LIN {X 0,Y 297.033,Z 357.775,A -85,B 0,C 180,E1 -16432.036,E2 -16432.036} C_VEL
LIN {X 0,Y 297.41,Z 355.086,A -85,B 0,C 180,E1 -16433.79,E2 -16433.79} C_VEL
LIN {X 0,Y 297.936,Z 351.345,A -85,B 0,C 180,E1 -16435.645,E2 -16435.645} C_VEL
LIN {X 0,Y 298.718,Z 345.55,A -85,B 0,C 180,E1 -16437.879,E2 -16437.879} C_VEL
LIN {X 0,Y 299.838,Z 337.982,A -85,B 0,C 180,E1 -16440.135,E2 -16440.135} C_VEL
LIN {X 0,Y 301.105,Z 329.348,A -85,B 0,C 180,E1 -16442.173,E2 -16442.173} C_VEL
LIN {X 0,Y 302.519,Z 319.297,A -85,B 0,C 180,E1 -16444.054,E2 -16444.054} C_VEL
LIN {X 0,Y 303.821,Z 309.214,A -85,B 0,C 180,E1 -16445.577,E2 -16445.577} C_VEL
LIN {X 0,Y 305.13,Z 297.791,A -85,B 0,C 180,E1 -16446.949,E2 -16446.949} C_VEL
LIN {X 0,Y 305.794,Z 291.875,A -85,B 0,C 180,E1 -16447.538,E2 -16447.538} C_VEL
LIN {X 0,Y 304.033,Z 282.592,A -85,B 0,C 180,E1 -16448.5,E2 -16448.5} C_VEL
LIN {X 0,Y 300.885,Z 269.635,A -85,B 0,C 180,E1 -16449.625,E2 -16449.625} C_VEL
LIN {X 0,Y 297.457,Z 257.519,A -85,B 0,C 180,E1 -16450.469,E2 -16450.469} C_VEL
LIN {X 0,Y 297.653,Z 253.673,A -85,B 0,C 180,E1 -16454.947,E2 -16454.947} C_VEL
LIN {X 0,Y 297.831,Z 251.39,A -85,B 0,C 180,E1 -16457.739,E2 -16457.739} C_VEL
LIN {X 0,Y 298.536,Z 251.297,A -85,B 0,C 180,E1 -16461.881,E2 -16461.881} C_VEL
LIN {X 0,Y 298.622,Z 251.286,A -85,B 0,C 180,E1 -16464.599,E2 -16464.599} C_VEL
LIN {X 0,Y 298.914,Z 251.25,A -85,B 0,C 180,E1 -16468.654,E2 -16468.654} C_VEL
LIN {X 0,Y 298.91,Z 251.253,A -85,B 0,C 180,E1 -16471.348,E2 -16471.348} C_VEL
LIN {X 0,Y 298.783,Z 251.266,A -85,B 0,C 180,E1 -16476.755,E2 -16476.755} C_VEL
LIN {X 0,Y 298.666,Z 251.281,A -85,B 0,C 180,E1 -16479.482,E2 -16479.482} C_VEL
LIN {X 0,Y 298.539,Z 251.297,A -85,B 0,C 180,E1 -16483.617,E2 -16483.617} C_VEL
LIN {X 0,Y 298.536,Z 251.297,A -85,B 0,C 180,E1 -16486.41,E2 -16486.41} C_VEL
LIN {X 0,Y 298.552,Z 251.294,A -85,B 0,C 180,E1 -16489.685,E2 -16489.685} C_VEL
LIN {X 0,Y 298.477,Z 251.304,A -85,B 0,C 180,E1 -16493.597,E2 -16493.597} C_VEL
LIN {X 0,Y 298.48,Z 251.305,A -85,B 0,C 180,E1 -16496.576,E2 -16496.576} C_VEL
LIN {X 0,Y 298.409,Z 251.311,A -85,B 0,C 180,E1 -16499.643,E2 -16499.643} C_VEL
LIN {X 0,Y 298.384,Z 251.319,A -85,B 0,C 180,E1 -16502.802,E2 -16502.802} C_VEL
LIN {X 0,Y 298.456,Z 251.308,A -85,B 0,C 180,E1 -16506.815,E2 -16506.815} C_VEL
LIN {X 0,Y 298.445,Z 251.307,A -85,B 0,C 180,E1 -16511.252,E2 -16511.252} C_VEL
LIN {X 0,Y 298.481,Z 251.302,A -85,B 0,C 180,E1 -16515.063,E2 -16515.063} C_VEL
LIN {X 0,Y 298.449,Z 251.306,A -85,B 0,C 180,E1 -16518.899,E2 -16518.899} C_VEL
LIN {X 0,Y 298.465,Z 251.304,A -85,B 0,C 180,E1 -16523.189,E2 -16523.189} C_VEL
LIN {X 0,Y 298.393,Z 251.312,A -85,B 0,C 180,E1 -16527.203,E2 -16527.203} C_VEL
LIN {X 0,Y 298.428,Z 251.309,A -85,B 0,C 180,E1 -16530.617,E2 -16530.617} C_VEL
LIN {X 0,Y 298.481,Z 251.302,A -85,B 0,C 180,E1 -16533.477,E2 -16533.477} C_VEL
LIN {X 0,Y 298.432,Z 251.309,A -85,B 0,C 180,E1 -16536.7,E2 -16536.7} C_VEL
LIN {X 0,Y 298.538,Z 251.293,A -85,B 0,C 180,E1 -16540.759,E2 -16540.759} C_VEL
LIN {X 0,Y 298.593,Z 251.287,A -85,B 0,C 180,E1 -16544.997,E2 -16544.997} C_VEL
LIN {X 0,Y 298.592,Z 251.289,A -85,B 0,C 180,E1 -16549.149,E2 -16549.149} C_VEL
LIN {X 0,Y 298.719,Z 251.277,A -85,B 0,C 180,E1 -16551.887,E2 -16551.887} C_VEL
LIN {X 0,Y 298.655,Z 251.278,A -85,B 0,C 180,E1 -16554.609,E2 -16554.609} C_VEL
LIN {X 0,Y 297.958,Z 251.369,A -85,B 0,C 180,E1 -16555.736,E2 -16555.736} C_VEL
LIN {X 0,Y 295.263,Z 251.704,A -85,B 0,C 180,E1 -16557.578,E2 -16557.578} C_VEL
LIN {X 0,Y 292.236,Z 252.085,A -85,B 0,C 180,E1 -16559.836,E2 -16559.836} C_VEL
LIN {X 0,Y 291.913,Z 252.12,A -85,B 0,C 180,E1 -16560.613,E2 -16560.613} C_VEL
LIN {X 0,Y 291.789,Z 252.136,A -85,B 0,C 180,E1 -16562.763,E2 -16562.763} C_VEL
LIN {X 0,Y 291.7,Z 252.144,A -85,B 0,C 180,E1 -16566.921,E2 -16566.921} C_VEL
LIN {X 0,Y 291.573,Z 252.167,A -85,B 0,C 180,E1 -16569.716,E2 -16569.716} C_VEL
LIN {X 0,Y 291.528,Z 252.169,A -85,B 0,C 180,E1 -16573.952,E2 -16573.952} C_VEL
LIN {X 0,Y 291.493,Z 252.171,A -85,B 0,C 180,E1 -16576.82,E2 -16576.82} C_VEL
LIN {X 0,Y 291.457,Z 252.179,A -85,B 0,C 180,E1 -16579.877,E2 -16579.877} C_VEL
LIN {X 0,Y 291.406,Z 252.184,A -85,B 0,C 180,E1 -16584.207,E2 -16584.207} C_VEL
LIN {X 0,Y 291.426,Z 252.186,A -85,B 0,C 180,E1 -16587.273,E2 -16587.273} C_VEL
LIN {X 0,Y 291.342,Z 252.192,A -85,B 0,C 180,E1 -16590.439,E2 -16590.439} C_VEL
LIN {X 0,Y 291.352,Z 252.192,A -85,B 0,C 180,E1 -16593.7,E2 -16593.7} C_VEL
LIN {X 0,Y 291.384,Z 252.191,A -85,B 0,C 180,E1 -16597.255,E2 -16597.255} C_VEL
LIN {X 0,Y 291.388,Z 252.232,A -85,B 0,C 180,E1 -16599.836,E2 -16599.836} C_VEL
LIN {X 0,Y 292.258,Z 257.11,A -85,B 0,C 180,E1 -16603.828,E2 -16603.828} C_VEL
LIN {X 0,Y 293.264,Z 262.494,A -85,B 0,C 180,E1 -16607.982,E2 -16607.982} C_VEL
LIN {X 0,Y 294.099,Z 267.529,A -85,B 0,C 180,E1 -16611.587,E2 -16611.587} C_VEL
LIN {X 0,Y 294.17,Z 270.073,A -85,B 0,C 180,E1 -16613.324,E2 -16613.324} C_VEL
LIN {X 0,Y 293.683,Z 273.84,A -85,B 0,C 180,E1 -16615.78,E2 -16615.78} C_VEL
LIN {X 0,Y 292.608,Z 280.296,A -85,B 0,C 180,E1 -16619.848,E2 -16619.848} C_VEL
LIN {X 0,Y 291.71,Z 286.456,A -85,B 0,C 180,E1 -16623.641,E2 -16623.641} C_VEL
LIN {X 0,Y 291.315,Z 289.802,A -85,B 0,C 180,E1 -16625.668,E2 -16625.668} C_VEL
LIN {X 0,Y 293.73,Z 303.932,A -85,B 0,C 180,E1 -16626.515,E2 -16626.515} C_VEL
LIN {X 0,Y 295.445,Z 316.454,A -85,B 0,C 180,E1 -16627.509,E2 -16627.509} C_VEL
LIN {X 0,Y 296.597,Z 328.112,A -85,B 0,C 180,E1 -16628.657,E2 -16628.657} C_VEL
LIN {X 0,Y 297.147,Z 337.485,A -85,B 0,C 180,E1 -16629.762,E2 -16629.762} C_VEL
LIN {X 0,Y 295.444,Z 348.79,A -85,B 0,C 180,E1 -16631.268,E2 -16631.268} C_VEL
LIN {X 0,Y 294.12,Z 358.492,A -85,B 0,C 180,E1 -16632.906,E2 -16632.906} C_VEL
LIN {X 0,Y 292.817,Z 367.103,A -85,B 0,C 180,E1 -16634.691,E2 -16634.691} C_VEL
LIN {X 0,Y 291.583,Z 375.192,A -85,B 0,C 180,E1 -16636.762,E2 -16636.762} C_VEL
LIN {X 0,Y 290.672,Z 381.694,A -85,B 0,C 180,E1 -16638.846,E2 -16638.846} C_VEL
LIN {X 0,Y 290.061,Z 386.848,A -85,B 0,C 180,E1 -16640.938,E2 -16640.938} C_VEL
LIN {X 0,Y 289.731,Z 390.835,A -85,B 0,C 180,E1 -16643.033,E2 -16643.033} C_VEL
LIN {X 0,Y 289.652,Z 392.878,A -85,B 0,C 180,E1 -16644.43,E2 -16644.43} C_VEL
LIN {X 0,Y 289.605,Z 394.493,A -85,B 0,C 180,E1 -16645.824,E2 -16645.824} C_VEL
LIN {X 0,Y 289.561,Z 395.692,A -85,B 0,C 180,E1 -16647.217,E2 -16647.217} C_VEL
LIN {X 0,Y 289.583,Z 396.449,A -85,B 0,C 180,E1 -16648.609,E2 -16648.609} C_VEL
LIN {X 0,Y 289.691,Z 396.79,A -85,B 0,C 180,E1 -16649.999,E2 -16649.999} C_VEL
LIN {X 0,Y 289.554,Z 396.262,A -85,B 0,C 180,E1 -16652.782,E2 -16652.782} C_VEL
LIN {X 0,Y 289.565,Z 395.378,A -85,B 0,C 180,E1 -16654.175,E2 -16654.175} C_VEL
LIN {X 0,Y 289.636,Z 393.816,A -85,B 0,C 180,E1 -16655.797,E2 -16655.797} C_VEL
LIN {X 0,Y 289.911,Z 390.214,A -85,B 0,C 180,E1 -16658.363,E2 -16658.363} C_VEL
LIN {X 0,Y 290.452,Z 386.109,A -85,B 0,C 180,E1 -16660.455,E2 -16660.455} C_VEL
LIN {X 0,Y 291.419,Z 379.871,A -85,B 0,C 180,E1 -16662.889,E2 -16662.889} C_VEL
LIN {X 0,Y 292.767,Z 373.132,A -85,B 0,C 180,E1 -16664.954,E2 -16664.954} C_VEL
LIN {X 0,Y 294.385,Z 364.544,A -85,B 0,C 180,E1 -16667.073,E2 -16667.073} C_VEL
LIN {X 0,Y 295.779,Z 356.408,A -85,B 0,C 180,E1 -16668.709,E2 -16668.709} C_VEL
LIN {X 0,Y 297.772,Z 346.112,A -85,B 0,C 180,E1 -16670.372,E2 -16670.372} C_VEL
LIN {X 0,Y 298.85,Z 338.795,A -85,B 0,C 180,E1 -16671.377,E2 -16671.377} C_VEL
LIN {X 0,Y 298.679,Z 327.3,A -85,B 0,C 180,E1 -16672.824,E2 -16672.824} C_VEL
LIN {X 0,Y 297.839,Z 315.601,A -85,B 0,C 180,E1 -16674.077,E2 -16674.077} C_VEL
LIN {X 0,Y 295.706,Z 302.829,A -85,B 0,C 180,E1 -16675.289,E2 -16675.289} C_VEL
LIN {X 0,Y 292.498,Z 290.386,A -85,B 0,C 180,E1 -16676.342,E2 -16676.342} C_VEL
LIN {X 0,Y 291.804,Z 287.336,A -85,B 0,C 180,E1 -16676.591,E2 -16676.591} C_VEL
LIN {X 0,Y 292.734,Z 281.581,A -85,B 0,C 180,E1 -16680.275,E2 -16680.275} C_VEL
LIN {X 0,Y 293.839,Z 275.714,A -85,B 0,C 180,E1 -16684.198,E2 -16684.198} C_VEL
LIN {X 0,Y 294.467,Z 272.269,A -85,B 0,C 180,E1 -16686.631,E2 -16686.631} C_VEL
LIN {X 0,Y 294.397,Z 268.901,A -85,B 0,C 180,E1 -16689.232,E2 -16689.232} C_VEL
LIN {X 0,Y 293.583,Z 264.391,A -85,B 0,C 180,E1 -16693.101,E2 -16693.101} C_VEL
LIN {X 0,Y 292.737,Z 259.678,A -85,B 0,C 180,E1 -16697.759,E2 -16697.759} C_VEL
LIN {X 0,Y 292.15,Z 256.569,A -85,B 0,C 180,E1 -16701.282,E2 -16701.282} C_VEL
LIN {X 0,Y 291.668,Z 253.761,A -85,B 0,C 180,E1 -16705.009,E2 -16705.009} C_VEL
LIN {X 0,Y 291.345,Z 252.195,A -85,B 0,C 180,E1 -16707.594,E2 -16707.594} C_VEL
LIN {X 0,Y 291.382,Z 252.187,A -85,B 0,C 180,E1 -16711.156,E2 -16711.156} C_VEL
LIN {X 0,Y 291.417,Z 252.186,A -85,B 0,C 180,E1 -16714.27,E2 -16714.27} C_VEL
LIN {X 0,Y 291.381,Z 252.185,A -85,B 0,C 180,E1 -16717.297,E2 -16717.297} C_VEL
LIN {X 0,Y 291.457,Z 252.176,A -85,B 0,C 180,E1 -16720.268,E2 -16720.268} C_VEL
LIN {X 0,Y 291.554,Z 252.164,A -85,B 0,C 180,E1 -16724.621,E2 -16724.621} C_VEL
LIN {X 0,Y 291.535,Z 252.168,A -85,B 0,C 180,E1 -16728.878,E2 -16728.878} C_VEL
LIN {X 0,Y 291.706,Z 252.146,A -85,B 0,C 180,E1 -16731.686,E2 -16731.686} C_VEL
LIN {X 0,Y 291.629,Z 252.16,A -85,B 0,C 180,E1 -16734.466,E2 -16734.466} C_VEL
LIN {X 0,Y 291.888,Z 252.129,A -85,B 0,C 180,E1 -16738.618,E2 -16738.618} C_VEL
LIN {X 0,Y 291.887,Z 252.126,A -85,B 0,C 180,E1 -16741.377,E2 -16741.377} C_VEL
LIN {X 0,Y 291.644,Z 252.357,A -85,B 0,C 180,E1 -16745.529,E2 -16745.529} C_VEL
LIN {X 0,Y 291.961,Z 253.705,A -85,B 0,C 180,E1 -16748.302,E2 -16748.302} C_VEL
LIN {X 0,Y 291.794,Z 256.101,A -85,B 0,C 180,E1 -16752.517,E2 -16752.517} C_VEL
LIN {X 0,Y 291.598,Z 257.897,A -85,B 0,C 180,E1 -16755.41,E2 -16755.41} C_VEL
LIN {X 0,Y 291.238,Z 260.78,A -85,B 0,C 180,E1 -16759.761,E2 -16759.761} C_VEL
LIN {X 0,Y 291.188,Z 261.337,A -85,B 0,C 180,E1 -16760.482,E2 -16760.482} C_VEL
LIN {X 0,Y 292.271,Z 264.393,A -85,B 0,C 180,E1 -16760.771,E2 -16760.771} C_VEL
LIN {X 0,Y 296.77,Z 275.63,A -85,B 0,C 180,E1 -16762.011,E2 -16762.011} C_VEL
LIN {X 0,Y 300.031,Z 286.603,A -85,B 0,C 180,E1 -16763.281,E2 -16763.281} C_VEL
LIN {X 0,Y 302.16,Z 296.713,A -85,B 0,C 180,E1 -16764.564,E2 -16764.564} C_VEL
LIN {X 0,Y 302.165,Z 299.449,A -85,B 0,C 180,E1 -16764.896,E2 -16764.896} C_VEL
LIN {X 0,Y 300.604,Z 309.905,A -85,B 0,C 180,E1 -16766.165,E2 -16766.165} C_VEL
LIN {X 0,Y 298.7,Z 320.617,A -85,B 0,C 180,E1 -16767.782,E2 -16767.782} C_VEL
LIN {X 0,Y 296.859,Z 330.143,A -85,B 0,C 180,E1 -16769.601,E2 -16769.601} C_VEL
LIN {X 0,Y 295.135,Z 338.506,A -85,B 0,C 180,E1 -16771.59,E2 -16771.59} C_VEL
LIN {X 0,Y 293.541,Z 345.871,A -85,B 0,C 180,E1 -16773.821,E2 -16773.821} C_VEL
LIN {X 0,Y 292.187,Z 351.715,A -85,B 0,C 180,E1 -16776.103,E2 -16776.103} C_VEL
LIN {X 0,Y 291.343,Z 355.527,A -85,B 0,C 180,E1 -16778.041,E2 -16778.041} C_VEL
LIN {X 0,Y 290.847,Z 357.596,A -85,B 0,C 180,E1 -16779.355,E2 -16779.355} C_VEL
LIN {X 0,Y 290.279,Z 359.966,A -85,B 0,C 180,E1 -16781.364,E2 -16781.364} C_VEL
LIN {X 0,Y 289.86,Z 361.443,A -85,B 0,C 180,E1 -16783.334,E2 -16783.334} C_VEL
LIN {X 0,Y 289.632,Z 362.114,A -85,B 0,C 180,E1 -16785.277,E2 -16785.277} C_VEL
LIN {X 0,Y 289.486,Z 362.005,A -85,B 0,C 180,E1 -16787.176,E2 -16787.176} C_VEL
LIN {X 0,Y 289.573,Z 361.135,A -85,B 0,C 180,E1 -16789.059,E2 -16789.059} C_VEL
LIN {X 0,Y 289.921,Z 358.545,A -85,B 0,C 180,E1 -16791.82,E2 -16791.82} C_VEL
LIN {X 0,Y 290.317,Z 355.666,A -85,B 0,C 180,E1 -16793.779,E2 -16793.779} C_VEL
LIN {X 0,Y 291.051,Z 350.63,A -85,B 0,C 180,E1 -16796.264,E2 -16796.264} C_VEL
LIN {X 0,Y 291.846,Z 344.907,A -85,B 0,C 180,E1 -16798.416,E2 -16798.416} C_VEL
LIN {X 0,Y 293.013,Z 337.475,A -85,B 0,C 180,E1 -16800.62,E2 -16800.62} C_VEL
LIN {X 0,Y 294.287,Z 328.968,A -85,B 0,C 180,E1 -16802.618,E2 -16802.618} C_VEL
LIN {X 0,Y 295.782,Z 318.782,A -85,B 0,C 180,E1 -16804.536,E2 -16804.536} C_VEL
LIN {X 0,Y 297.178,Z 308.303,A -85,B 0,C 180,E1 -16806.11,E2 -16806.11} C_VEL
LIN {X 0,Y 298.568,Z 296.305,A -85,B 0,C 180,E1 -16807.538,E2 -16807.538} C_VEL
LIN {X 0,Y 298.958,Z 292.63,A -85,B 0,C 180,E1 -16807.907,E2 -16807.907} C_VEL
LIN {X 0,Y 296.84,Z 282.192,A -85,B 0,C 180,E1 -16809.017,E2 -16809.017} C_VEL
LIN {X 0,Y 293.698,Z 269.415,A -85,B 0,C 180,E1 -16810.149,E2 -16810.149} C_VEL
LIN {X 0,Y 290.453,Z 257.903,A -85,B 0,C 180,E1 -16810.984,E2 -16810.984} C_VEL
LIN {X 0,Y 290.637,Z 254.275,A -85,B 0,C 180,E1 -16815.284,E2 -16815.284} C_VEL
LIN {X 0,Y 290.749,Z 252.496,A -85,B 0,C 180,E1 -16817.436,E2 -16817.436} C_VEL
LIN {X 0,Y 291.433,Z 252.185,A -85,B 0,C 180,E1 -16821.367,E2 -16821.367} C_VEL
LIN {X 0,Y 291.617,Z 252.161,A -85,B 0,C 180,E1 -16823.08,E2 -16823.08} C_VEL
LIN {X 0,Y 291.783,Z 252.142,A -85,B 0,C 180,E1 -16827.24,E2 -16827.24} C_VEL
LIN {X 0,Y 291.965,Z 252.115,A -85,B 0,C 180,E1 -16830.001,E2 -16830.001} C_VEL
LIN {X 0,Y 291.776,Z 252.139,A -85,B 0,C 180,E1 -16832.762,E2 -16832.762} C_VEL
LIN {X 0,Y 291.732,Z 252.146,A -85,B 0,C 180,E1 -16836.919,E2 -16836.919} C_VEL
LIN {X 0,Y 291.615,Z 252.159,A -85,B 0,C 180,E1 -16839.713,E2 -16839.713} C_VEL
LIN {X 0,Y 291.509,Z 252.172,A -85,B 0,C 180,E1 -16843.952,E2 -16843.952} C_VEL
LIN {X 0,Y 291.475,Z 252.18,A -85,B 0,C 180,E1 -16846.819,E2 -16846.819} C_VEL
LIN {X 0,Y 291.482,Z 252.174,A -85,B 0,C 180,E1 -16849.901,E2 -16849.901} C_VEL
LIN {X 0,Y 291.425,Z 252.183,A -85,B 0,C 180,E1 -16854.204,E2 -16854.204} C_VEL
LIN {X 0,Y 291.414,Z 252.183,A -85,B 0,C 180,E1 -16857.273,E2 -16857.273} C_VEL
LIN {X 0,Y 291.326,Z 252.196,A -85,B 0,C 180,E1 -16860.439,E2 -16860.439} C_VEL
LIN {X 0,Y 291.334,Z 252.192,A -85,B 0,C 180,E1 -16863.7,E2 -16863.7} C_VEL
LIN {X 0,Y 291.389,Z 252.185,A -85,B 0,C 180,E1 -16867.262,E2 -16867.262} C_VEL
LIN {X 0,Y 291.392,Z 252.19,A -85,B 0,C 180,E1 -16870.633,E2 -16870.633} C_VEL
LIN {X 0,Y 291.399,Z 252.188,A -85,B 0,C 180,E1 -16874.382,E2 -16874.382} C_VEL
LIN {X 0,Y 291.384,Z 252.187,A -85,B 0,C 180,E1 -16878.392,E2 -16878.392} C_VEL
LIN {X 0,Y 291.381,Z 252.186,A -85,B 0,C 180,E1 -16881.167,E2 -16881.167} C_VEL
LIN {X 0,Y 291.381,Z 252.189,A -85,B 0,C 180,E1 -16884.632,E2 -16884.632} C_VEL
LIN {X 0,Y 291.371,Z 252.188,A -85,B 0,C 180,E1 -16887.954,E2 -16887.954} C_VEL
LIN {X 0,Y 291.378,Z 252.184,A -85,B 0,C 180,E1 -16891.161,E2 -16891.161} C_VEL
LIN {X 0,Y 291.414,Z 252.187,A -85,B 0,C 180,E1 -16894.275,E2 -16894.275} C_VEL
LIN {X 0,Y 291.379,Z 252.187,A -85,B 0,C 180,E1 -16897.302,E2 -16897.302} C_VEL
LIN {X 0,Y 291.457,Z 252.178,A -85,B 0,C 180,E1 -16900.273,E2 -16900.273} C_VEL
LIN {X 0,Y 291.555,Z 252.164,A -85,B 0,C 180,E1 -16904.626,E2 -16904.626} C_VEL
LIN {X 0,Y 291.536,Z 252.167,A -85,B 0,C 180,E1 -16908.883,E2 -16908.883} C_VEL
LIN {X 0,Y 291.669,Z 252.154,A -85,B 0,C 180,E1 -16911.69,E2 -16911.69} C_VEL
LIN {X 0,Y 291.613,Z 252.154,A -85,B 0,C 180,E1 -16914.581,E2 -16914.581} C_VEL
LIN {X 0,Y 291.892,Z 252.122,A -85,B 0,C 180,E1 -16918.623,E2 -16918.623} C_VEL
LIN {X 0,Y 291.913,Z 252.12,A -85,B 0,C 180,E1 -16920.613,E2 -16920.613} C_VEL
LIN {X 0,Y 291.166,Z 252.218,A -85,B 0,C 180,E1 -16921.762,E2 -16921.762} C_VEL
LIN {X 0,Y 288.165,Z 252.591,A -85,B 0,C 180,E1 -16923.628,E2 -16923.628} C_VEL
LIN {X 0,Y 285.685,Z 252.896,A -85,B 0,C 180,E1 -16925.144,E2 -16925.144} C_VEL
LIN {X 0,Y 284.674,Z 253.019,A -85,B 0,C 180,E1 -16926.321,E2 -16926.321} C_VEL
LIN {X 0,Y 284.619,Z 253.025,A -85,B 0,C 180,E1 -16926.72,E2 -16926.72} C_VEL
LIN {X 0,Y 284.519,Z 253.043,A -85,B 0,C 180,E1 -16929.959,E2 -16929.959} C_VEL
LIN {X 0,Y 284.487,Z 253.045,A -85,B 0,C 180,E1 -16934.305,E2 -16934.305} C_VEL
LIN {X 0,Y 284.431,Z 253.053,A -85,B 0,C 180,E1 -16937.25,E2 -16937.25} C_VEL
LIN {X 0,Y 284.385,Z 253.058,A -85,B 0,C 180,E1 -16940.244,E2 -16940.244} C_VEL
LIN {X 0,Y 284.376,Z 253.061,A -85,B 0,C 180,E1 -16943.877,E2 -16943.877} C_VEL
LIN {X 0,Y 284.401,Z 253.06,A -85,B 0,C 180,E1 -16947.174,E2 -16947.174} C_VEL
LIN {X 0,Y 284.301,Z 253.074,A -85,B 0,C 180,E1 -16951.276,E2 -16951.276} C_VEL
LIN {X 0,Y 284.349,Z 253.067,A -85,B 0,C 180,E1 -16955.349,E2 -16955.349} C_VEL
LIN {X 0,Y 284.371,Z 253.254,A -85,B 0,C 180,E1 -16959.526,E2 -16959.526} C_VEL
LIN {X 0,Y 284.973,Z 256.48,A -85,B 0,C 180,E1 -16962.28,E2 -16962.28} C_VEL
LIN {X 0,Y 285.89,Z 261.734,A -85,B 0,C 180,E1 -16966.502,E2 -16966.502} C_VEL
LIN {X 0,Y 286.641,Z 265.615,A -85,B 0,C 180,E1 -16969.473,E2 -16969.473} C_VEL
LIN {X 0,Y 287.147,Z 269.515,A -85,B 0,C 180,E1 -16972.274,E2 -16972.274} C_VEL
LIN {X 0,Y 286.841,Z 273.283,A -85,B 0,C 180,E1 -16974.845,E2 -16974.845} C_VEL
LIN {X 0,Y 285.642,Z 280.374,A -85,B 0,C 180,E1 -16979.449,E2 -16979.449} C_VEL
LIN {X 0,Y 284.627,Z 286.96,A -85,B 0,C 180,E1 -16983.611,E2 -16983.611} C_VEL
LIN {X 0,Y 284.3,Z 289.426,A -85,B 0,C 180,E1 -16985.149,E2 -16985.149} C_VEL
LIN {X 0,Y 286.806,Z 303.726,A -85,B 0,C 180,E1 -16986.031,E2 -16986.031} C_VEL
LIN {X 0,Y 288.498,Z 316.349,A -85,B 0,C 180,E1 -16987.059,E2 -16987.059} C_VEL
LIN {X 0,Y 289.712,Z 328.742,A -85,B 0,C 180,E1 -16988.329,E2 -16988.329} C_VEL
LIN {X 0,Y 290.098,Z 339.197,A -85,B 0,C 180,E1 -16989.619,E2 -16989.619} C_VEL
LIN {X 0,Y 288.361,Z 350.006,A -85,B 0,C 180,E1 -16991.159,E2 -16991.159} C_VEL
LIN {X 0,Y 286.932,Z 359.778,A -85,B 0,C 180,E1 -16992.906,E2 -16992.906} C_VEL
LIN {X 0,Y 285.666,Z 367.804,A -85,B 0,C 180,E1 -16994.664,E2 -16994.664} C_VEL
LIN {X 0,Y 284.428,Z 375.68,A -85,B 0,C 180,E1 -16996.787,E2 -16996.787} C_VEL
LIN {X 0,Y 283.642,Z 381.026,A -85,B 0,C 180,E1 -16998.566,E2 -16998.566} C_VEL
LIN {X 0,Y 283.039,Z 386.242,A -85,B 0,C 180,E1 -17000.711,E2 -17000.711} C_VEL
LIN {X 0,Y 282.67,Z 390.273,A -85,B 0,C 180,E1 -17002.858,E2 -17002.858} C_VEL
LIN {X 0,Y 282.573,Z 392.345,A -85,B 0,C 180,E1 -17004.29,E2 -17004.29} C_VEL
LIN {X 0,Y 282.525,Z 393.98,A -85,B 0,C 180,E1 -17005.719,E2 -17005.719} C_VEL
LIN {X 0,Y 282.488,Z 395.199,A -85,B 0,C 180,E1 -17007.147,E2 -17007.147} C_VEL
LIN {X 0,Y 282.498,Z 395.993,A -85,B 0,C 180,E1 -17008.574,E2 -17008.574} C_VEL
LIN {X 0,Y 282.602,Z 396.352,A -85,B 0,C 180,E1 -17009.999,E2 -17009.999} C_VEL
LIN {X 0,Y 282.48,Z 395.859,A -85,B 0,C 180,E1 -17012.851,E2 -17012.851} C_VEL
LIN {X 0,Y 282.486,Z 395.009,A -85,B 0,C 180,E1 -17014.28,E2 -17014.28} C_VEL
LIN {X 0,Y 282.529,Z 393.716,A -85,B 0,C 180,E1 -17015.71,E2 -17015.71} C_VEL
LIN {X 0,Y 282.744,Z 391.024,A -85,B 0,C 180,E1 -17017.857,E2 -17017.857} C_VEL
LIN {X 0,Y 283.2,Z 387.329,A -85,B 0,C 180,E1 -17020.003,E2 -17020.003} C_VEL
LIN {X 0,Y 283.94,Z 382.545,A -85,B 0,C 180,E1 -17022.144,E2 -17022.144} C_VEL
LIN {X 0,Y 285.386,Z 375.411,A -85,B 0,C 180,E1 -17024.62,E2 -17024.62} C_VEL
LIN {X 0,Y 286.948,Z 367.754,A -85,B 0,C 180,E1 -17026.724,E2 -17026.724} C_VEL
LIN {X 0,Y 288.404,Z 359.993,A -85,B 0,C 180,E1 -17028.468,E2 -17028.468} C_VEL
LIN {X 0,Y 290.469,Z 349.552,A -85,B 0,C 180,E1 -17030.352,E2 -17030.352} C_VEL
LIN {X 0,Y 292.129,Z 340.36,A -85,B 0,C 180,E1 -17031.708,E2 -17031.708} C_VEL
LIN {X 0,Y 292.141,Z 328.287,A -85,B 0,C 180,E1 -17033.325,E2 -17033.325} C_VEL
LIN {X 0,Y 291.507,Z 317.905,A -85,B 0,C 180,E1 -17034.51,E2 -17034.51} C_VEL
LIN {X 0,Y 289.633,Z 305.544,A -85,B 0,C 180,E1 -17035.768,E2 -17035.768} C_VEL
LIN {X 0,Y 286.667,Z 293.298,A -85,B 0,C 180,E1 -17036.9,E2 -17036.9} C_VEL
LIN {X 0,Y 284.969,Z 286.853,A -85,B 0,C 180,E1 -17037.455,E2 -17037.455} C_VEL
LIN {X 0,Y 286.139,Z 280.206,A -85,B 0,C 180,E1 -17041.874,E2 -17041.874} C_VEL
LIN {X 0,Y 287.311,Z 274.427,A -85,B 0,C 180,E1 -17045.948,E2 -17045.948} C_VEL
LIN {X 0,Y 287.486,Z 271.079,A -85,B 0,C 180,E1 -17048.527,E2 -17048.527} C_VEL
LIN {X 0,Y 286.962,Z 267.729,A -85,B 0,C 180,E1 -17051.395,E2 -17051.395} C_VEL
LIN {X 0,Y 286.306,Z 264.28,A -85,B 0,C 180,E1 -17054.611,E2 -17054.611} C_VEL
LIN {X 0,Y 285.698,Z 260.651,A -85,B 0,C 180,E1 -17058.378,E2 -17058.378} C_VEL
LIN {X 0,Y 285.129,Z 257.579,A -85,B 0,C 180,E1 -17062.067,E2 -17062.067} C_VEL
LIN {X 0,Y 284.703,Z 255.207,A -85,B 0,C 180,E1 -17065.403,E2 -17065.403} C_VEL
LIN {X 0,Y 284.315,Z 253.21,A -85,B 0,C 180,E1 -17068.726,E2 -17068.726} C_VEL
LIN {X 0,Y 284.332,Z 253.07,A -85,B 0,C 180,E1 -17071.987,E2 -17071.987} C_VEL
LIN {X 0,Y 284.347,Z 253.067,A -85,B 0,C 180,E1 -17075.152,E2 -17075.152} C_VEL
LIN {X 0,Y 284.327,Z 253.066,A -85,B 0,C 180,E1 -17078.235,E2 -17078.235} C_VEL
LIN {X 0,Y 284.403,Z 253.058,A -85,B 0,C 180,E1 -17081.259,E2 -17081.259} C_VEL
LIN {X 0,Y 284.491,Z 253.044,A -85,B 0,C 180,E1 -17084.457,E2 -17084.457} C_VEL
LIN {X 0,Y 284.486,Z 253.047,A -85,B 0,C 180,E1 -17088.599,E2 -17088.599} C_VEL
LIN {X 0,Y 284.656,Z 253.024,A -85,B 0,C 180,E1 -17091.479,E2 -17091.479} C_VEL
LIN {X 0,Y 284.599,Z 253.034,A -85,B 0,C 180,E1 -17094.329,E2 -17094.329} C_VEL
LIN {X 0,Y 284.853,Z 253.005,A -85,B 0,C 180,E1 -17098.584,E2 -17098.584} C_VEL
LIN {X 0,Y 284.853,Z 253.002,A -85,B 0,C 180,E1 -17101.411,E2 -17101.411} C_VEL
LIN {X 0,Y 284.524,Z 253.192,A -85,B 0,C 180,E1 -17104.247,E2 -17104.247} C_VEL
LIN {X 0,Y 284.902,Z 254.443,A -85,B 0,C 180,E1 -17107.082,E2 -17107.082} C_VEL
LIN {X 0,Y 284.912,Z 255.927,A -85,B 0,C 180,E1 -17109.941,E2 -17109.941} C_VEL
LIN {X 0,Y 284.787,Z 257.554,A -85,B 0,C 180,E1 -17112.83,E2 -17112.83} C_VEL
LIN {X 0,Y 284.559,Z 259.337,A -85,B 0,C 180,E1 -17115.761,E2 -17115.761} C_VEL
LIN {X 0,Y 284.273,Z 261.863,A -85,B 0,C 180,E1 -17119.607,E2 -17119.607} C_VEL
LIN {X 0,Y 285.366,Z 264.961,A -85,B 0,C 180,E1 -17119.92,E2 -17119.92} C_VEL
LIN {X 0,Y 289.842,Z 275.814,A -85,B 0,C 180,E1 -17121.186,E2 -17121.186} C_VEL
LIN {X 0,Y 293.256,Z 286.87,A -85,B 0,C 180,E1 -17122.544,E2 -17122.544} C_VEL
LIN {X 0,Y 295.621,Z 298.038,A -85,B 0,C 180,E1 -17124.021,E2 -17124.021} C_VEL
LIN {X 0,Y 295.834,Z 299.917,A -85,B 0,C 180,E1 -17124.283,E2 -17124.283} C_VEL
LIN {X 0,Y 294.097,Z 311.014,A -85,B 0,C 180,E1 -17125.663,E2 -17125.663} C_VEL
LIN {X 0,Y 292.248,Z 320.843,A -85,B 0,C 180,E1 -17127.185,E2 -17127.185} C_VEL
LIN {X 0,Y 290.407,Z 329.937,A -85,B 0,C 180,E1 -17128.945,E2 -17128.945} C_VEL
LIN {X 0,Y 288.481,Z 338.737,A -85,B 0,C 180,E1 -17131.066,E2 -17131.066} C_VEL
LIN {X 0,Y 286.97,Z 345.293,A -85,B 0,C 180,E1 -17133.041,E2 -17133.041} C_VEL
LIN {X 0,Y 285.684,Z 350.566,A -85,B 0,C 180,E1 -17135.022,E2 -17135.022} C_VEL
LIN {X 0,Y 284.662,Z 354.755,A -85,B 0,C 180,E1 -17137.015,E2 -17137.015} C_VEL
LIN {X 0,Y 283.904,Z 357.944,A -85,B 0,C 180,E1 -17138.997,E2 -17138.997} C_VEL
LIN {X 0,Y 283.549,Z 359.367,A -85,B 0,C 180,E1 -17140.119,E2 -17140.119} C_VEL
LIN {X 0,Y 283.021,Z 361.223,A -85,B 0,C 180,E1 -17142.099,E2 -17142.099} C_VEL
LIN {X 0,Y 282.672,Z 362.308,A -85,B 0,C 180,E1 -17144.115,E2 -17144.115} C_VEL
LIN {X 0,Y 282.468,Z 362.598,A -85,B 0,C 180,E1 -17146.177,E2 -17146.177} C_VEL
LIN {X 0,Y 282.425,Z 362.007,A -85,B 0,C 180,E1 -17148.286,E2 -17148.286} C_VEL
LIN {X 0,Y 282.613,Z 360.489,A -85,B 0,C 180,E1 -17150.43,E2 -17150.43} C_VEL
LIN {X 0,Y 282.996,Z 357.965,A -85,B 0,C 180,E1 -17152.622,E2 -17152.622} C_VEL
LIN {X 0,Y 283.617,Z 353.528,A -85,B 0,C 180,E1 -17155.255,E2 -17155.255} C_VEL
LIN {X 0,Y 284.45,Z 348.128,A -85,B 0,C 180,E1 -17157.595,E2 -17157.595} C_VEL
LIN {X 0,Y 285.572,Z 340.799,A -85,B 0,C 180,E1 -17160.049,E2 -17160.049} C_VEL
LIN {X 0,Y 286.914,Z 332.262,A -85,B 0,C 180,E1 -17162.264,E2 -17162.264} C_VEL
LIN {X 0,Y 288.354,Z 322.921,A -85,B 0,C 180,E1 -17164.209,E2 -17164.209} C_VEL
LIN {X 0,Y 289.851,Z 312.465,A -85,B 0,C 180,E1 -17165.943,E2 -17165.943} C_VEL
LIN {X 0,Y 291.36,Z 300.782,A -85,B 0,C 180,E1 -17167.486,E2 -17167.486} C_VEL
LIN {X 0,Y 292.093,Z 293.369,A -85,B 0,C 180,E1 -17168.289,E2 -17168.289} C_VEL
LIN {X 0,Y 289.538,Z 281.139,A -85,B 0,C 180,E1 -17169.623,E2 -17169.623} C_VEL
LIN {X 0,Y 286.311,Z 268.56,A -85,B 0,C 180,E1 -17170.749,E2 -17170.749} C_VEL
LIN {X 0,Y 283.392,Z 258.298,A -85,B 0,C 180,E1 -17171.521,E2 -17171.521} C_VEL
LIN {X 0,Y 283.619,Z 254.856,A -85,B 0,C 180,E1 -17175.654,E2 -17175.654} C_VEL
LIN {X 0,Y 283.681,Z 253.669,A -85,B 0,C 180,E1 -17177.117,E2 -17177.117} C_VEL
LIN {X 0,Y 283.877,Z 253.126,A -85,B 0,C 180,E1 -17178.577,E2 -17178.577} C_VEL
LIN {X 0,Y 284.424,Z 253.058,A -85,B 0,C 180,E1 -17181.475,E2 -17181.475} C_VEL
LIN {X 0,Y 284.551,Z 253.039,A -85,B 0,C 180,E1 -17184.331,E2 -17184.331} C_VEL
LIN {X 0,Y 284.846,Z 253.002,A -85,B 0,C 180,E1 -17188.587,E2 -17188.587} C_VEL
LIN {X 0,Y 284.842,Z 253.005,A -85,B 0,C 180,E1 -17191.415,E2 -17191.415} C_VEL
LIN {X 0,Y 284.684,Z 253.024,A -85,B 0,C 180,E1 -17197.091,E2 -17197.091} C_VEL
LIN {X 0,Y 284.553,Z 253.038,A -85,B 0,C 180,E1 -17199.957,E2 -17199.957} C_VEL
LIN {X 0,Y 284.469,Z 253.049,A -85,B 0,C 180,E1 -17204.304,E2 -17204.304} C_VEL
LIN {X 0,Y 284.416,Z 253.057,A -85,B 0,C 180,E1 -17207.25,E2 -17207.25} C_VEL
LIN {X 0,Y 284.413,Z 253.055,A -85,B 0,C 180,E1 -17210.24,E2 -17210.24} C_VEL
LIN {X 0,Y 284.385,Z 253.059,A -85,B 0,C 180,E1 -17213.89,E2 -17213.89} C_VEL
LIN {X 0,Y 284.323,Z 253.065,A -85,B 0,C 180,E1 -17218.012,E2 -17218.012} C_VEL
LIN {X 0,Y 284.284,Z 253.073,A -85,B 0,C 180,E1 -17221.276,E2 -17221.276} C_VEL
LIN {X 0,Y 284.351,Z 253.06,A -85,B 0,C 180,E1 -17225.356,E2 -17225.356} C_VEL
LIN {X 0,Y 284.322,Z 253.065,A -85,B 0,C 180,E1 -17228.168,E2 -17228.168} C_VEL
LIN {X 0,Y 284.344,Z 253.065,A -85,B 0,C 180,E1 -17232.145,E2 -17232.145} C_VEL
LIN {X 0,Y 284.346,Z 253.064,A -85,B 0,C 180,E1 -17236.211,E2 -17236.211} C_VEL
LIN {X 0,Y 284.345,Z 253.063,A -85,B 0,C 180,E1 -17240.016,E2 -17240.016} C_VEL
LIN {X 0,Y 284.35,Z 253.063,A -85,B 0,C 180,E1 -17243.62,E2 -17243.62} C_VEL
LIN {X 0,Y 284.304,Z 253.066,A -85,B 0,C 180,E1 -17247.192,E2 -17247.192} C_VEL
LIN {X 0,Y 284.355,Z 253.062,A -85,B 0,C 180,E1 -17250.379,E2 -17250.379} C_VEL
LIN {X 0,Y 284.375,Z 253.059,A -85,B 0,C 180,E1 -17253.589,E2 -17253.589} C_VEL
LIN {X 0,Y 284.364,Z 253.062,A -85,B 0,C 180,E1 -17256.71,E2 -17256.71} C_VEL
LIN {X 0,Y 284.402,Z 253.053,A -85,B 0,C 180,E1 -17261.264,E2 -17261.264} C_VEL
LIN {X 0,Y 284.492,Z 253.044,A -85,B 0,C 180,E1 -17264.462,E2 -17264.462} C_VEL
LIN {X 0,Y 284.488,Z 253.046,A -85,B 0,C 180,E1 -17268.604,E2 -17268.604} C_VEL
LIN {X 0,Y 284.623,Z 253.03,A -85,B 0,C 180,E1 -17271.483,E2 -17271.483} C_VEL
LIN {X 0,Y 284.595,Z 253.029,A -85,B 0,C 180,E1 -17274.334,E2 -17274.334} C_VEL
LIN {X 0,Y 284.858,Z 252.998,A -85,B 0,C 180,E1 -17278.589,E2 -17278.589} C_VEL
LIN {X 0,Y 284.857,Z 253.002,A -85,B 0,C 180,E1 -17281.416,E2 -17281.416} C_VEL
LIN {X 0,Y 284.619,Z 253.025,A -85,B 0,C 180,E1 -17286.72,E2 -17286.72} C_VEL
LIN {X 0,Y 284.345,Z 253.063,A -85,B 0,C 180,E1 -17287.509,E2 -17287.509} C_VEL
LIN {X 0,Y 282.993,Z 253.233,A -85,B 0,C 180,E1 -17288.673,E2 -17288.673} C_VEL
LIN {X 0,Y 278.544,Z 253.789,A -85,B 0,C 180,E1 -17291.377,E2 -17291.377} C_VEL
LIN {X 0,Y 277.485,Z 253.918,A -85,B 0,C 180,E1 -17292.588,E2 -17292.588} C_VEL
LIN {X 0,Y 277.413,Z 253.928,A -85,B 0,C 180,E1 -17292.999,E2 -17292.999} C_VEL
LIN {X 0,Y 277.412,Z 253.924,A -85,B 0,C 180,E1 -17296.183,E2 -17296.183} C_VEL
LIN {X 0,Y 277.352,Z 253.934,A -85,B 0,C 180,E1 -17300.352,E2 -17300.352} C_VEL
LIN {X 0,Y 277.325,Z 253.938,A -85,B 0,C 180,E1 -17304.172,E2 -17304.172} C_VEL
LIN {X 0,Y 277.33,Z 253.941,A -85,B 0,C 180,E1 -17307.505,E2 -17307.505} C_VEL
LIN {X 0,Y 277.28,Z 253.944,A -85,B 0,C 180,E1 -17310.483,E2 -17310.483} C_VEL
LIN {X 0,Y 277.254,Z 253.948,A -85,B 0,C 180,E1 -17313.897,E2 -17313.897} C_VEL
LIN {X 0,Y 277.276,Z 253.948,A -85,B 0,C 180,E1 -17317.47,E2 -17317.47} C_VEL
LIN {X 0,Y 277.299,Z 254.038,A -85,B 0,C 180,E1 -17319.009,E2 -17319.009} C_VEL
LIN {X 0,Y 278.127,Z 258.662,A -85,B 0,C 180,E1 -17323.023,E2 -17323.023} C_VEL
LIN {X 0,Y 279.059,Z 263.71,A -85,B 0,C 180,E1 -17327.157,E2 -17327.157} C_VEL
LIN {X 0,Y 279.764,Z 267.619,A -85,B 0,C 180,E1 -17330.164,E2 -17330.164} C_VEL
LIN {X 0,Y 280.102,Z 271.483,A -85,B 0,C 180,E1 -17332.973,E2 -17332.973} C_VEL
LIN {X 0,Y 279.409,Z 276.052,A -85,B 0,C 180,E1 -17336.107,E2 -17336.107} C_VEL
LIN {X 0,Y 278.255,Z 282.676,A -85,B 0,C 180,E1 -17340.493,E2 -17340.493} C_VEL
LIN {X 0,Y 277.312,Z 289.176,A -85,B 0,C 180,E1 -17344.617,E2 -17344.617} C_VEL
LIN {X 0,Y 279.718,Z 302.677,A -85,B 0,C 180,E1 -17345.468,E2 -17345.468} C_VEL
LIN {X 0,Y 281.525,Z 316.044,A -85,B 0,C 180,E1 -17346.587,E2 -17346.587} C_VEL
LIN {X 0,Y 282.768,Z 328.814,A -85,B 0,C 180,E1 -17347.932,E2 -17347.932} C_VEL
LIN {X 0,Y 283.211,Z 339.417,A -85,B 0,C 180,E1 -17349.29,E2 -17349.29} C_VEL
LIN {X 0,Y 281.427,Z 350.095,A -85,B 0,C 180,E1 -17350.866,E2 -17350.866} C_VEL
LIN {X 0,Y 279.858,Z 360.373,A -85,B 0,C 180,E1 -17352.773,E2 -17352.773} C_VEL
LIN {X 0,Y 278.517,Z 368.473,A -85,B 0,C 180,E1 -17354.635,E2 -17354.635} C_VEL
LIN {X 0,Y 277.276,Z 376.095,A -85,B 0,C 180,E1 -17356.813,E2 -17356.813} C_VEL
LIN {X 0,Y 276.393,Z 382.229,A -85,B 0,C 180,E1 -17359.005,E2 -17359.005} C_VEL
LIN {X 0,Y 275.829,Z 387.083,A -85,B 0,C 180,E1 -17361.206,E2 -17361.206} C_VEL
LIN {X 0,Y 275.531,Z 390.794,A -85,B 0,C 180,E1 -17363.408,E2 -17363.408} C_VEL
LIN {X 0,Y 275.447,Z 393.463,A -85,B 0,C 180,E1 -17365.609,E2 -17365.609} C_VEL
LIN {X 0,Y 275.418,Z 394.702,A -85,B 0,C 180,E1 -17367.074,E2 -17367.074} C_VEL
LIN {X 0,Y 275.416,Z 395.53,A -85,B 0,C 180,E1 -17368.537,E2 -17368.537} C_VEL
LIN {X 0,Y 275.513,Z 395.912,A -85,B 0,C 180,E1 -17369.999,E2 -17369.999} C_VEL
LIN {X 0,Y 275.408,Z 395.46,A -85,B 0,C 180,E1 -17372.925,E2 -17372.925} C_VEL
LIN {X 0,Y 275.428,Z 393.617,A -85,B 0,C 180,E1 -17375.63,E2 -17375.63} C_VEL
LIN {X 0,Y 275.684,Z 390.736,A -85,B 0,C 180,E1 -17378.059,E2 -17378.059} C_VEL
LIN {X 0,Y 276.185,Z 387.088,A -85,B 0,C 180,E1 -17380.26,E2 -17380.26} C_VEL
LIN {X 0,Y 276.963,Z 382.354,A -85,B 0,C 180,E1 -17382.455,E2 -17382.455} C_VEL
LIN {X 0,Y 278.509,Z 375.275,A -85,B 0,C 180,E1 -17384.989,E2 -17384.989} C_VEL
LIN {X 0,Y 280.144,Z 367.701,A -85,B 0,C 180,E1 -17387.143,E2 -17387.143} C_VEL
LIN {X 0,Y 281.652,Z 360.051,A -85,B 0,C 180,E1 -17388.927,E2 -17388.927} C_VEL
LIN {X 0,Y 283.61,Z 350.861,A -85,B 0,C 180,E1 -17390.677,E2 -17390.677} C_VEL
LIN {X 0,Y 285.412,Z 342.009,A -85,B 0,C 180,E1 -17392.055,E2 -17392.055} C_VEL
LIN {X 0,Y 285.578,Z 330.403,A -85,B 0,C 180,E1 -17393.7,E2 -17393.7} C_VEL
LIN {X 0,Y 285.149,Z 320.208,A -85,B 0,C 180,E1 -17394.941,E2 -17394.941} C_VEL
LIN {X 0,Y 283.553,Z 308.25,A -85,B 0,C 180,E1 -17396.261,E2 -17396.261} C_VEL
LIN {X 0,Y 280.883,Z 296.303,A -85,B 0,C 180,E1 -17397.461,E2 -17397.461} C_VEL
LIN {X 0,Y 278.205,Z 287.085,A -85,B 0,C 180,E1 -17398.308,E2 -17398.308} C_VEL
LIN {X 0,Y 278.13,Z 286.323,A -85,B 0,C 180,E1 -17398.388,E2 -17398.388} C_VEL
LIN {X 0,Y 279.305,Z 280.034,A -85,B 0,C 180,E1 -17402.75,E2 -17402.75} C_VEL
LIN {X 0,Y 280.102,Z 276.582,A -85,B 0,C 180,E1 -17405.245,E2 -17405.245} C_VEL
LIN {X 0,Y 280.496,Z 273.19,A -85,B 0,C 180,E1 -17407.868,E2 -17407.868} C_VEL
LIN {X 0,Y 280.135,Z 269.858,A -85,B 0,C 180,E1 -17410.713,E2 -17410.713} C_VEL
LIN {X 0,Y 279.674,Z 267.17,A -85,B 0,C 180,E1 -17413.216,E2 -17413.216} C_VEL
LIN {X 0,Y 278.965,Z 263.347,A -85,B 0,C 180,E1 -17417.137,E2 -17417.137} C_VEL
LIN {X 0,Y 278.392,Z 260.143,A -85,B 0,C 180,E1 -17420.864,E2 -17420.864} C_VEL
LIN {X 0,Y 277.947,Z 257.516,A -85,B 0,C 180,E1 -17424.437,E2 -17424.437} C_VEL
LIN {X 0,Y 277.515,Z 255.411,A -85,B 0,C 180,E1 -17427.869,E2 -17427.869} C_VEL
LIN {X 0,Y 277.272,Z 253.944,A -85,B 0,C 180,E1 -17431.208,E2 -17431.208} C_VEL
LIN {X 0,Y 277.314,Z 253.942,A -85,B 0,C 180,E1 -17434.477,E2 -17434.477} C_VEL
LIN {X 0,Y 277.285,Z 253.94,A -85,B 0,C 180,E1 -17437.653,E2 -17437.653} C_VEL
LIN {X 0,Y 277.345,Z 253.937,A -85,B 0,C 180,E1 -17440.764,E2 -17440.764} C_VEL
LIN {X 0,Y 277.433,Z 253.926,A -85,B 0,C 180,E1 -17445.324,E2 -17445.324} C_VEL
LIN {X 0,Y 277.504,Z 253.916,A -85,B 0,C 180,E1 -17449.786,E2 -17449.786} C_VEL
LIN {X 0,Y 277.651,Z 253.901,A -85,B 0,C 180,E1 -17452.727,E2 -17452.727} C_VEL
LIN {X 0,Y 277.819,Z 253.88,A -85,B 0,C 180,E1 -17458.548,E2 -17458.548} C_VEL
LIN {X 0,Y 277.818,Z 253.878,A -85,B 0,C 180,E1 -17461.447,E2 -17461.447} C_VEL
LIN {X 0,Y 277.697,Z 254.029,A -85,B 0,C 180,E1 -17462.899,E2 -17462.899} C_VEL
LIN {X 0,Y 277.94,Z 255.913,A -85,B 0,C 180,E1 -17467.261,E2 -17467.261} C_VEL
LIN {X 0,Y 277.925,Z 257.382,A -85,B 0,C 180,E1 -17470.193,E2 -17470.193} C_VEL
LIN {X 0,Y 277.763,Z 259.018,A -85,B 0,C 180,E1 -17473.16,E2 -17473.16} C_VEL
LIN {X 0,Y 277.512,Z 260.808,A -85,B 0,C 180,E1 -17476.172,E2 -17476.172} C_VEL
LIN {X 0,Y 277.326,Z 262.477,A -85,B 0,C 180,E1 -17478.657,E2 -17478.657} C_VEL
LIN {X 0,Y 278.37,Z 265.365,A -85,B 0,C 180,E1 -17478.966,E2 -17478.966} C_VEL
LIN {X 0,Y 282.523,Z 275.065,A -85,B 0,C 180,E1 -17480.184,E2 -17480.184} C_VEL
LIN {X 0,Y 286.208,Z 286.078,A -85,B 0,C 180,E1 -17481.61,E2 -17481.61} C_VEL
LIN {X 0,Y 288.714,Z 296.972,A -85,B 0,C 180,E1 -17483.109,E2 -17483.109} C_VEL
LIN {X 0,Y 289.348,Z 301.877,A -85,B 0,C 180,E1 -17483.813,E2 -17483.813} C_VEL
LIN {X 0,Y 287.48,Z 312.818,A -85,B 0,C 180,E1 -17485.241,E2 -17485.241} C_VEL
LIN {X 0,Y 285.51,Z 322.593,A -85,B 0,C 180,E1 -17486.836,E2 -17486.836} C_VEL
LIN {X 0,Y 283.449,Z 332.105,A -85,B 0,C 180,E1 -17488.773,E2 -17488.773} C_VEL
LIN {X 0,Y 281.628,Z 339.941,A -85,B 0,C 180,E1 -17490.766,E2 -17490.766} C_VEL
LIN {X 0,Y 279.844,Z 347.18,A -85,B 0,C 180,E1 -17493.105,E2 -17493.105} C_VEL
LIN {X 0,Y 278.352,Z 352.931,A -85,B 0,C 180,E1 -17495.497,E2 -17495.497} C_VEL
LIN {X 0,Y 277.131,Z 357.671,A -85,B 0,C 180,E1 -17498.174,E2 -17498.174} C_VEL
LIN {X 0,Y 276.421,Z 360.318,A -85,B 0,C 180,E1 -17500.295,E2 -17500.295} C_VEL
LIN {X 0,Y 275.888,Z 362.029,A -85,B 0,C 180,E1 -17502.376,E2 -17502.376} C_VEL
LIN {X 0,Y 275.542,Z 362.886,A -85,B 0,C 180,E1 -17504.426,E2 -17504.426} C_VEL
LIN {X 0,Y 275.369,Z 362.976,A -85,B 0,C 180,E1 -17506.443,E2 -17506.443} C_VEL
LIN {X 0,Y 275.341,Z 362.345,A -85,B 0,C 180,E1 -17508.423,E2 -17508.423} C_VEL
LIN {X 0,Y 275.528,Z 360.955,A -85,B 0,C 180,E1 -17510.382,E2 -17510.382} C_VEL
LIN {X 0,Y 276.023,Z 357.571,A -85,B 0,C 180,E1 -17513.249,E2 -17513.249} C_VEL
LIN {X 0,Y 276.792,Z 352.6,A -85,B 0,C 180,E1 -17516.042,E2 -17516.042} C_VEL
LIN {X 0,Y 277.582,Z 347.367,A -85,B 0,C 180,E1 -17518.235,E2 -17518.235} C_VEL
LIN {X 0,Y 278.75,Z 340.293,A -85,B 0,C 180,E1 -17520.552,E2 -17520.552} C_VEL
LIN {X 0,Y 280.122,Z 331.851,A -85,B 0,C 180,E1 -17522.751,E2 -17522.751} C_VEL
LIN {X 0,Y 281.596,Z 322.417,A -85,B 0,C 180,E1 -17524.717,E2 -17524.717} C_VEL
LIN {X 0,Y 283.116,Z 312.296,A -85,B 0,C 180,E1 -17526.405,E2 -17526.405} C_VEL
LIN {X 0,Y 284.563,Z 301.367,A -85,B 0,C 180,E1 -17527.875,E2 -17527.875} C_VEL
LIN {X 0,Y 285.173,Z 294.203,A -85,B 0,C 180,E1 -17528.685,E2 -17528.685} C_VEL
LIN {X 0,Y 282.753,Z 282.421,A -85,B 0,C 180,E1 -17530.017,E2 -17530.017} C_VEL
LIN {X 0,Y 279.509,Z 269.658,A -85,B 0,C 180,E1 -17531.207,E2 -17531.207} C_VEL
LIN {X 0,Y 276.371,Z 258.713,A -85,B 0,C 180,E1 -17532.042,E2 -17532.042} C_VEL
LIN {X 0,Y 276.541,Z 256.072,A -85,B 0,C 180,E1 -17535.278,E2 -17535.278} C_VEL
LIN {X 0,Y 276.759,Z 254.014,A -85,B 0,C 180,E1 -17538.28,E2 -17538.28} C_VEL
LIN {X 0,Y 277.34,Z 253.94,A -85,B 0,C 180,E1 -17541.255,E2 -17541.255} C_VEL
LIN {X 0,Y 277.514,Z 253.916,A -85,B 0,C 180,E1 -17544.187,E2 -17544.187} C_VEL
LIN {X 0,Y 277.811,Z 253.879,A -85,B 0,C 180,E1 -17548.551,E2 -17548.551} C_VEL
LIN {X 0,Y 277.808,Z 253.881,A -85,B 0,C 180,E1 -17551.45,E2 -17551.45} C_VEL
LIN {X 0,Y 277.639,Z 253.902,A -85,B 0,C 180,E1 -17557.272,E2 -17557.272} C_VEL
LIN {X 0,Y 277.493,Z 253.917,A -85,B 0,C 180,E1 -17560.213,E2 -17560.213} C_VEL
LIN {X 0,Y 277.421,Z 253.929,A -85,B 0,C 180,E1 -17564.676,E2 -17564.676} C_VEL
LIN {X 0,Y 277.364,Z 253.936,A -85,B 0,C 180,E1 -17569.233,E2 -17569.233} C_VEL
LIN {X 0,Y 277.365,Z 253.934,A -85,B 0,C 180,E1 -17573.918,E2 -17573.918} C_VEL
LIN {X 0,Y 277.316,Z 253.938,A -85,B 0,C 180,E1 -17577.508,E2 -17577.508} C_VEL
LIN {X 0,Y 277.261,Z 253.949,A -85,B 0,C 180,E1 -17580.483,E2 -17580.483} C_VEL
LIN {X 0,Y 277.244,Z 253.948,A -85,B 0,C 180,E1 -17583.897,E2 -17583.897} C_VEL
LIN {X 0,Y 277.276,Z 253.941,A -85,B 0,C 180,E1 -17587.469,E2 -17587.469} C_VEL
LIN {X 0,Y 277.287,Z 253.943,A -85,B 0,C 180,E1 -17591.223,E2 -17591.223} C_VEL
LIN {X 0,Y 277.28,Z 253.941,A -85,B 0,C 180,E1 -17595.211,E2 -17595.211} C_VEL
LIN {X 0,Y 277.289,Z 253.94,A -85,B 0,C 180,E1 -17599.497,E2 -17599.497} C_VEL
LIN {X 0,Y 277.285,Z 253.946,A -85,B 0,C 180,E1 -17602.537,E2 -17602.537} C_VEL
LIN {X 0,Y 277.25,Z 253.95,A -85,B 0,C 180,E1 -17606.108,E2 -17606.108} C_VEL
LIN {X 0,Y 277.257,Z 253.941,A -85,B 0,C 180,E1 -17609.541,E2 -17609.541} C_VEL
LIN {X 0,Y 277.356,Z 253.933,A -85,B 0,C 180,E1 -17612.867,E2 -17612.867} C_VEL
LIN {X 0,Y 277.327,Z 253.941,A -85,B 0,C 180,E1 -17616.082,E2 -17616.082} C_VEL
LIN {X 0,Y 277.344,Z 253.932,A -85,B 0,C 180,E1 -17620.769,E2 -17620.769} C_VEL
LIN {X 0,Y 277.434,Z 253.922,A -85,B 0,C 180,E1 -17625.329,E2 -17625.329} C_VEL
LIN {X 0,Y 277.461,Z 253.924,A -85,B 0,C 180,E1 -17629.79,E2 -17629.79} C_VEL
LIN {X 0,Y 277.63,Z 253.898,A -85,B 0,C 180,E1 -17632.731,E2 -17632.731} C_VEL
LIN {X 0,Y 277.824,Z 253.875,A -85,B 0,C 180,E1 -17638.553,E2 -17638.553} C_VEL
LIN {X 0,Y 277.823,Z 253.878,A -85,B 0,C 180,E1 -17641.452,E2 -17641.452} C_VEL
LIN {X 0,Y 277.613,Z 253.899,A -85,B 0,C 180,E1 -17647.274,E2 -17647.274} C_VEL
LIN {X 0,Y 277.462,Z 253.921,A -85,B 0,C 180,E1 -17650.215,E2 -17650.215} C_VEL
LIN {X 0,Y 277.413,Z 253.928,A -85,B 0,C 180,E1 -17652.999,E2 -17652.999} C_VEL
LIN {X 0,Y 276.764,Z 254.011,A -85,B 0,C 180,E1 -17654.211,E2 -17654.211} C_VEL
LIN {X 0,Y 273.854,Z 254.37,A -85,B 0,C 180,E1 -17656.182,E2 -17656.182} C_VEL
LIN {X 0,Y 271.384,Z 254.679,A -85,B 0,C 180,E1 -17657.785,E2 -17657.785} C_VEL
LIN {X 0,Y 270.356,Z 254.807,A -85,B 0,C 180,E1 -17659.029,E2 -17659.029} C_VEL
LIN {X 0,Y 270.29,Z 254.814,A -85,B 0,C 180,E1 -17659.45,E2 -17659.45} C_VEL
LIN {X 0,Y 270.284,Z 254.815,A -85,B 0,C 180,E1 -17664.482,E2 -17664.482} C_VEL
LIN {X 0,Y 270.277,Z 254.817,A -85,B 0,C 180,E1 -17667.91,E2 -17667.91} C_VEL
LIN {X 0,Y 270.192,Z 254.831,A -85,B 0,C 180,E1 -17671.35,E2 -17671.35} C_VEL
LIN {X 0,Y 270.21,Z 254.828,A -85,B 0,C 180,E1 -17674.907,E2 -17674.907} C_VEL
LIN {X 0,Y 270.285,Z 254.969,A -85,B 0,C 180,E1 -17678.615,E2 -17678.615} C_VEL
LIN {X 0,Y 271.012,Z 259.186,A -85,B 0,C 180,E1 -17682.398,E2 -17682.398} C_VEL
LIN {X 0,Y 271.861,Z 263.912,A -85,B 0,C 180,E1 -17686.375,E2 -17686.375} C_VEL
LIN {X 0,Y 272.69,Z 268.311,A -85,B 0,C 180,E1 -17689.884,E2 -17689.884} C_VEL
LIN {X 0,Y 273.079,Z 272.358,A -85,B 0,C 180,E1 -17692.926,E2 -17692.926} C_VEL
LIN {X 0,Y 272.497,Z 276.176,A -85,B 0,C 180,E1 -17695.624,E2 -17695.624} C_VEL
LIN {X 0,Y 271.396,Z 282.104,A -85,B 0,C 180,E1 -17699.67,E2 -17699.67} C_VEL
LIN {X 0,Y 270.346,Z 288.603,A -85,B 0,C 180,E1 -17704.019,E2 -17704.019} C_VEL
LIN {X 0,Y 272.828,Z 302.947,A -85,B 0,C 180,E1 -17704.977,E2 -17704.977} C_VEL
LIN {X 0,Y 274.659,Z 316.393,A -85,B 0,C 180,E1 -17706.157,E2 -17706.157} C_VEL
LIN {X 0,Y 275.836,Z 328.92,A -85,B 0,C 180,E1 -17707.53,E2 -17707.53} C_VEL
LIN {X 0,Y 276.289,Z 339.506,A -85,B 0,C 180,E1 -17708.942,E2 -17708.942} C_VEL
LIN {X 0,Y 274.512,Z 350.104,A -85,B 0,C 180,E1 -17710.559,E2 -17710.559} C_VEL
LIN {X 0,Y 272.854,Z 360.402,A -85,B 0,C 180,E1 -17712.532,E2 -17712.532} C_VEL
LIN {X 0,Y 271.647,Z 367.621,A -85,B 0,C 180,E1 -17714.237,E2 -17714.237} C_VEL
LIN {X 0,Y 270.352,Z 375.34,A -85,B 0,C 180,E1 -17716.469,E2 -17716.469} C_VEL
LIN {X 0,Y 269.378,Z 381.532,A -85,B 0,C 180,E1 -17718.715,E2 -17718.715} C_VEL
LIN {X 0,Y 268.798,Z 386.446,A -85,B 0,C 180,E1 -17720.974,E2 -17720.974} C_VEL
LIN {X 0,Y 268.463,Z 390.21,A -85,B 0,C 180,E1 -17723.234,E2 -17723.234} C_VEL
LIN {X 0,Y 268.373,Z 392.93,A -85,B 0,C 180,E1 -17725.493,E2 -17725.493} C_VEL
LIN {X 0,Y 268.348,Z 394.194,A -85,B 0,C 180,E1 -17726.997,E2 -17726.997} C_VEL
LIN {X 0,Y 268.336,Z 395.049,A -85,B 0,C 180,E1 -17728.498,E2 -17728.498} C_VEL
LIN {X 0,Y 268.426,Z 395.471,A -85,B 0,C 180,E1 -17729.999,E2 -17729.999} C_VEL
LIN {X 0,Y 268.336,Z 395.063,A -85,B 0,C 180,E1 -17733.002,E2 -17733.002} C_VEL
LIN {X 0,Y 268.349,Z 393.422,A -85,B 0,C 180,E1 -17735.593,E2 -17735.593} C_VEL
LIN {X 0,Y 268.616,Z 390.443,A -85,B 0,C 180,E1 -17738.273,E2 -17738.273} C_VEL
LIN {X 0,Y 269.164,Z 386.837,A -85,B 0,C 180,E1 -17740.53,E2 -17740.53} C_VEL
LIN {X 0,Y 270.005,Z 382.173,A -85,B 0,C 180,E1 -17742.781,E2 -17742.781} C_VEL
LIN {X 0,Y 271.644,Z 375.194,A -85,B 0,C 180,E1 -17745.377,E2 -17745.377} C_VEL
LIN {X 0,Y 273.354,Z 367.705,A -85,B 0,C 180,E1 -17747.583,E2 -17747.583} C_VEL
LIN {X 0,Y 275.278,Z 358.484,A -85,B 0,C 180,E1 -17749.771,E2 -17749.771} C_VEL
LIN {X 0,Y 277.678,Z 347.949,A -85,B 0,C 180,E1 -17751.724,E2 -17751.724} C_VEL
LIN {X 0,Y 278.777,Z 342.346,A -85,B 0,C 180,E1 -17752.609,E2 -17752.609} C_VEL
LIN {X 0,Y 279.09,Z 330.172,A -85,B 0,C 180,E1 -17754.403,E2 -17754.403} C_VEL
LIN {X 0,Y 278.556,Z 319.512,A -85,B 0,C 180,E1 -17755.767,E2 -17755.767} C_VEL
LIN {X 0,Y 277.052,Z 308.559,A -85,B 0,C 180,E1 -17757.036,E2 -17757.036} C_VEL
LIN {X 0,Y 274.247,Z 296.117,A -85,B 0,C 180,E1 -17758.361,E2 -17758.361} C_VEL
LIN {X 0,Y 271.425,Z 286.667,A -85,B 0,C 180,E1 -17759.31,E2 -17759.31} C_VEL
LIN {X 0,Y 271.34,Z 285.79,A -85,B 0,C 180,E1 -17759.385,E2 -17759.385} C_VEL
LIN {X 0,Y 272.537,Z 279.91,A -85,B 0,C 180,E1 -17763.644,E2 -17763.644} C_VEL
LIN {X 0,Y 273.303,Z 276.457,A -85,B 0,C 180,E1 -17766.258,E2 -17766.258} C_VEL
LIN {X 0,Y 273.518,Z 274.209,A -85,B 0,C 180,E1 -17768.072,E2 -17768.072} C_VEL
LIN {X 0,Y 273.282,Z 272,A -85,B 0,C 180,E1 -17770.009,E2 -17770.009} C_VEL
LIN {X 0,Y 272.597,Z 268.035,A -85,B 0,C 180,E1 -17773.787,E2 -17773.787} C_VEL
LIN {X 0,Y 271.803,Z 263.636,A -85,B 0,C 180,E1 -17778.576,E2 -17778.576} C_VEL
LIN {X 0,Y 271.387,Z 261.239,A -85,B 0,C 180,E1 -17781.57,E2 -17781.57} C_VEL
LIN {X 0,Y 270.925,Z 258.709,A -85,B 0,C 180,E1 -17785.199,E2 -17785.199} C_VEL
LIN {X 0,Y 270.517,Z 256.499,A -85,B 0,C 180,E1 -17789.017,E2 -17789.017} C_VEL
LIN {X 0,Y 270.304,Z 255.062,A -85,B 0,C 180,E1 -17792.128,E2 -17792.128} C_VEL
LIN {X 0,Y 270.277,Z 254.818,A -85,B 0,C 180,E1 -17795.517,E2 -17795.517} C_VEL
LIN {X 0,Y 270.301,Z 254.811,A -85,B 0,C 180,E1 -17800.242,E2 -17800.242} C_VEL
LIN {X 0,Y 270.401,Z 254.799,A -85,B 0,C 180,E1 -17804.933,E2 -17804.933} C_VEL
LIN {X 0,Y 270.44,Z 254.795,A -85,B 0,C 180,E1 -17809.517,E2 -17809.517} C_VEL
LIN {X 0,Y 270.609,Z 254.779,A -85,B 0,C 180,E1 -17812.536,E2 -17812.536} C_VEL
LIN {X 0,Y 270.785,Z 254.756,A -85,B 0,C 180,E1 -17818.51,E2 -17818.51} C_VEL
LIN {X 0,Y 270.792,Z 254.954,A -85,B 0,C 180,E1 -17821.485,E2 -17821.485} C_VEL
LIN {X 0,Y 270.976,Z 257.387,A -85,B 0,C 180,E1 -17827.448,E2 -17827.448} C_VEL
LIN {X 0,Y 270.937,Z 258.853,A -85,B 0,C 180,E1 -17830.459,E2 -17830.459} C_VEL
LIN {X 0,Y 270.725,Z 260.514,A -85,B 0,C 180,E1 -17833.509,E2 -17833.509} C_VEL
LIN {X 0,Y 270.385,Z 262.88,A -85,B 0,C 180,E1 -17837.585,E2 -17837.585} C_VEL
LIN {X 0,Y 271.563,Z 266.084,A -85,B 0,C 180,E1 -17837.992,E2 -17837.992} C_VEL
LIN {X 0,Y 275.49,Z 274.971,A -85,B 0,C 180,E1 -17839.183,E2 -17839.183} C_VEL
LIN {X 0,Y 279.215,Z 285.437,A -85,B 0,C 180,E1 -17840.631,E2 -17840.631} C_VEL
LIN {X 0,Y 282.124,Z 297.47,A -85,B 0,C 180,E1 -17842.363,E2 -17842.363} C_VEL
LIN {X 0,Y 282.971,Z 303.204,A -85,B 0,C 180,E1 -17843.23,E2 -17843.23} C_VEL
LIN {X 0,Y 280.916,Z 314.458,A -85,B 0,C 180,E1 -17844.772,E2 -17844.772} C_VEL
LIN {X 0,Y 278.647,Z 325.054,A -85,B 0,C 180,E1 -17846.6,E2 -17846.6} C_VEL
LIN {X 0,Y 276.588,Z 333.956,A -85,B 0,C 180,E1 -17848.538,E2 -17848.538} C_VEL
LIN {X 0,Y 274.518,Z 342.22,A -85,B 0,C 180,E1 -17850.795,E2 -17850.795} C_VEL
LIN {X 0,Y 273.037,Z 347.861,A -85,B 0,C 180,E1 -17852.717,E2 -17852.717} C_VEL
LIN {X 0,Y 271.732,Z 352.54,A -85,B 0,C 180,E1 -17854.677,E2 -17854.677} C_VEL
LIN {X 0,Y 270.702,Z 356.315,A -85,B 0,C 180,E1 -17856.661,E2 -17856.661} C_VEL
LIN {X 0,Y 269.864,Z 359.277,A -85,B 0,C 180,E1 -17858.68,E2 -17858.68} C_VEL
LIN {X 0,Y 269.193,Z 361.476,A -85,B 0,C 180,E1 -17860.791,E2 -17860.791} C_VEL
LIN {X 0,Y 268.701,Z 362.865,A -85,B 0,C 180,E1 -17862.917,E2 -17862.917} C_VEL
LIN {X 0,Y 268.404,Z 363.453,A -85,B 0,C 180,E1 -17865.012,E2 -17865.012} C_VEL
LIN {X 0,Y 268.263,Z 363.249,A -85,B 0,C 180,E1 -17867.18,E2 -17867.18} C_VEL
LIN {X 0,Y 268.326,Z 362.144,A -85,B 0,C 180,E1 -17869.421,E2 -17869.421} C_VEL
LIN {X 0,Y 268.64,Z 360.069,A -85,B 0,C 180,E1 -17871.701,E2 -17871.701} C_VEL
LIN {X 0,Y 269.133,Z 356.902,A -85,B 0,C 180,E1 -17874.043,E2 -17874.043} C_VEL
LIN {X 0,Y 269.963,Z 351.528,A -85,B 0,C 180,E1 -17876.86,E2 -17876.86} C_VEL
LIN {X 0,Y 271.004,Z 345.271,A -85,B 0,C 180,E1 -17879.329,E2 -17879.329} C_VEL
LIN {X 0,Y 272.122,Z 338.624,A -85,B 0,C 180,E1 -17881.408,E2 -17881.408} C_VEL
LIN {X 0,Y 273.619,Z 329.734,A -85,B 0,C 180,E1 -17883.629,E2 -17883.629} C_VEL
LIN {X 0,Y 275.133,Z 320.57,A -85,B 0,C 180,E1 -17885.476,E2 -17885.476} C_VEL
LIN {X 0,Y 276.512,Z 311.115,A -85,B 0,C 180,E1 -17887.036,E2 -17887.036} C_VEL
LIN {X 0,Y 278.089,Z 299.36,A -85,B 0,C 180,E1 -17888.582,E2 -17888.582} C_VEL
LIN {X 0,Y 278.42,Z 296.101,A -85,B 0,C 180,E1 -17888.958,E2 -17888.958} C_VEL
LIN {X 0,Y 276.292,Z 285.11,A -85,B 0,C 180,E1 -17890.265,E2 -17890.265} C_VEL
LIN {X 0,Y 273.15,Z 272.399,A -85,B 0,C 180,E1 -17891.532,E2 -17891.532} C_VEL
LIN {X 0,Y 269.325,Z 259.097,A -85,B 0,C 180,E1 -17892.636,E2 -17892.636} C_VEL
LIN {X 0,Y 269.538,Z 256.069,A -85,B 0,C 180,E1 -17896.429,E2 -17896.429} C_VEL
LIN {X 0,Y 269.667,Z 254.897,A -85,B 0,C 180,E1 -17897.967,E2 -17897.967} C_VEL
LIN {X 0,Y 270.264,Z 254.821,A -85,B 0,C 180,E1 -17901.152,E2 -17901.152} C_VEL
LIN {X 0,Y 270.478,Z 254.793,A -85,B 0,C 180,E1 -17904.035,E2 -17904.035} C_VEL
LIN {X 0,Y 270.777,Z 254.755,A -85,B 0,C 180,E1 -17908.514,E2 -17908.514} C_VEL
LIN {X 0,Y 270.774,Z 254.757,A -85,B 0,C 180,E1 -17911.488,E2 -17911.488} C_VEL
LIN {X 0,Y 270.597,Z 254.778,A -85,B 0,C 180,E1 -17917.462,E2 -17917.462} C_VEL
LIN {X 0,Y 270.428,Z 254.798,A -85,B 0,C 180,E1 -17920.482,E2 -17920.482} C_VEL
LIN {X 0,Y 270.39,Z 254.808,A -85,B 0,C 180,E1 -17925.066,E2 -17925.066} C_VEL
LIN {X 0,Y 270.318,Z 254.811,A -85,B 0,C 180,E1 -17929.755,E2 -17929.755} C_VEL
LIN {X 0,Y 270.28,Z 254.819,A -85,B 0,C 180,E1 -17934.586,E2 -17934.586} C_VEL
LIN {X 0,Y 270.261,Z 254.816,A -85,B 0,C 180,E1 -17937.911,E2 -17937.911} C_VEL
LIN {X 0,Y 270.173,Z 254.83,A -85,B 0,C 180,E1 -17941.35,E2 -17941.35} C_VEL
LIN {X 0,Y 270.205,Z 254.824,A -85,B 0,C 180,E1 -17944.906,E2 -17944.906} C_VEL
LIN {X 0,Y 270.213,Z 254.827,A -85,B 0,C 180,E1 -17948.719,E2 -17948.719} C_VEL
LIN {X 0,Y 270.252,Z 254.823,A -85,B 0,C 180,E1 -17952.543,E2 -17952.543} C_VEL
LIN {X 0,Y 270.225,Z 254.818,A -85,B 0,C 180,E1 -17956.738,E2 -17956.738} C_VEL
LIN {X 0,Y 270.242,Z 254.817,A -85,B 0,C 180,E1 -17959.451,E2 -17959.451} C_VEL
LIN {X 0,Y 270.252,Z 254.819,A -85,B 0,C 180,E1 -17963.724,E2 -17963.724} C_VEL
LIN {X 0,Y 270.2,Z 254.824,A -85,B 0,C 180,E1 -17966.896,E2 -17966.896} C_VEL
LIN {X 0,Y 270.217,Z 254.821,A -85,B 0,C 180,E1 -17970.389,E2 -17970.389} C_VEL
LIN {X 0,Y 270.261,Z 254.817,A -85,B 0,C 180,E1 -17973.767,E2 -17973.767} C_VEL
LIN {X 0,Y 270.231,Z 254.821,A -85,B 0,C 180,E1 -17977.042,E2 -17977.042} C_VEL
LIN {X 0,Y 270.3,Z 254.812,A -85,B 0,C 180,E1 -17980.247,E2 -17980.247} C_VEL
LIN {X 0,Y 270.403,Z 254.797,A -85,B 0,C 180,E1 -17984.938,E2 -17984.938} C_VEL
LIN {X 0,Y 270.413,Z 254.8,A -85,B 0,C 180,E1 -17989.521,E2 -17989.521} C_VEL
LIN {X 0,Y 270.586,Z 254.775,A -85,B 0,C 180,E1 -17992.541,E2 -17992.541} C_VEL
LIN {X 0,Y 270.79,Z 254.751,A -85,B 0,C 180,E1 -17998.515,E2 -17998.515} C_VEL
LIN {X 0,Y 270.789,Z 254.755,A -85,B 0,C 180,E1 -18001.49,E2 -18001.49} C_VEL
LIN {X 0,Y 270.573,Z 254.777,A -85,B 0,C 180,E1 -18007.465,E2 -18007.465} C_VEL
LIN {X 0,Y 270.415,Z 254.798,A -85,B 0,C 180,E1 -18010.484,E2 -18010.484} C_VEL
LIN {X 0,Y 270.409,Z 254.799,A -85,B 0,C 180,E1 -18015.067,E2 -18015.067} C_VEL
LIN {X 0,Y 270.29,Z 254.814,A -85,B 0,C 180,E1 -18019.45,E2 -18019.45} C_VEL
LIN {X 0,Y 269.663,Z 254.898,A -85,B 0,C 180,E1 -18020.694,E2 -18020.694} C_VEL
LIN {X 0,Y 266.798,Z 255.258,A -85,B 0,C 180,E1 -18022.719,E2 -18022.719} C_VEL
LIN {X 0,Y 264.333,Z 255.561,A -85,B 0,C 180,E1 -18024.367,E2 -18024.367} C_VEL
LIN {X 0,Y 263.267,Z 255.692,A -85,B 0,C 180,E1 -18025.644,E2 -18025.644} C_VEL
LIN {X 0,Y 263.178,Z 255.7,A -85,B 0,C 180,E1 -18026.078,E2 -18026.078} C_VEL
LIN {X 0,Y 263.173,Z 255.702,A -85,B 0,C 180,E1 -18028.733,E2 -18028.733} C_VEL
LIN {X 0,Y 263.14,Z 255.706,A -85,B 0,C 180,E1 -18032.29,E2 -18032.29} C_VEL
LIN {X 0,Y 263.191,Z 255.702,A -85,B 0,C 180,E1 -18036.765,E2 -18036.765} C_VEL
LIN {X 0,Y 263.228,Z 255.793,A -85,B 0,C 180,E1 -18038.128,E2 -18038.128} C_VEL
LIN {X 0,Y 263.901,Z 259.748,A -85,B 0,C 180,E1 -18041.782,E2 -18041.782} C_VEL
LIN {X 0,Y 264.728,Z 264.334,A -85,B 0,C 180,E1 -18045.793,E2 -18045.793} C_VEL
LIN {X 0,Y 265.386,Z 267.673,A -85,B 0,C 180,E1 -18048.542,E2 -18048.542} C_VEL
LIN {X 0,Y 265.966,Z 271.538,A -85,B 0,C 180,E1 -18051.603,E2 -18051.603} C_VEL
LIN {X 0,Y 265.911,Z 274.09,A -85,B 0,C 180,E1 -18053.51,E2 -18053.51} C_VEL
LIN {X 0,Y 265.239,Z 277.8,A -85,B 0,C 180,E1 -18056.19,E2 -18056.19} C_VEL
LIN {X 0,Y 264.104,Z 283.967,A -85,B 0,C 180,E1 -18060.507,E2 -18060.507} C_VEL
LIN {X 0,Y 263.416,Z 288.434,A -85,B 0,C 180,E1 -18063.466,E2 -18063.466} C_VEL
LIN {X 0,Y 265.838,Z 302.222,A -85,B 0,C 180,E1 -18064.394,E2 -18064.394} C_VEL
LIN {X 0,Y 267.651,Z 315.618,A -85,B 0,C 180,E1 -18065.592,E2 -18065.592} C_VEL
LIN {X 0,Y 268.782,Z 327.395,A -85,B 0,C 180,E1 -18066.907,E2 -18066.907} C_VEL
LIN {X 0,Y 269.324,Z 338.26,A -85,B 0,C 180,E1 -18068.37,E2 -18068.37} C_VEL
LIN {X 0,Y 268.835,Z 343.391,A -85,B 0,C 180,E1 -18069.133,E2 -18069.133} C_VEL
LIN {X 0,Y 267.102,Z 353.178,A -85,B 0,C 180,E1 -18070.797,E2 -18070.797} C_VEL
LIN {X 0,Y 265.629,Z 362.105,A -85,B 0,C 180,E1 -18072.674,E2 -18072.674} C_VEL
LIN {X 0,Y 264.065,Z 370.895,A -85,B 0,C 180,E1 -18074.959,E2 -18074.959} C_VEL
LIN {X 0,Y 262.812,Z 377.877,A -85,B 0,C 180,E1 -18077.254,E2 -18077.254} C_VEL
LIN {X 0,Y 261.941,Z 384.287,A -85,B 0,C 180,E1 -18079.956,E2 -18079.956} C_VEL
LIN {X 0,Y 261.494,Z 388.477,A -85,B 0,C 180,E1 -18082.276,E2 -18082.276} C_VEL
LIN {X 0,Y 261.352,Z 391.202,A -85,B 0,C 180,E1 -18084.265,E2 -18084.265} C_VEL
LIN {X 0,Y 261.281,Z 393.684,A -85,B 0,C 180,E1 -18086.915,E2 -18086.915} C_VEL
LIN {X 0,Y 261.259,Z 394.563,A -85,B 0,C 180,E1 -18088.458,E2 -18088.458} C_VEL
LIN {X 0,Y 261.341,Z 395.03,A -85,B 0,C 180,E1 -18089.999,E2 -18089.999} C_VEL
LIN {X 0,Y 261.253,Z 395.043,A -85,B 0,C 180,E1 -18091.541,E2 -18091.541} C_VEL
LIN {X 0,Y 261.265,Z 394.665,A -85,B 0,C 180,E1 -18093.083,E2 -18093.083} C_VEL
LIN {X 0,Y 261.302,Z 392.721,A -85,B 0,C 180,E1 -18096.175,E2 -18096.175} C_VEL
LIN {X 0,Y 261.566,Z 390.157,A -85,B 0,C 180,E1 -18098.497,E2 -18098.497} C_VEL
LIN {X 0,Y 262.134,Z 386.607,A -85,B 0,C 180,E1 -18100.816,E2 -18100.816} C_VEL
LIN {X 0,Y 263.066,Z 382.004,A -85,B 0,C 180,E1 -18103.125,E2 -18103.125} C_VEL
LIN {X 0,Y 264.79,Z 375.123,A -85,B 0,C 180,E1 -18105.786,E2 -18105.786} C_VEL
LIN {X 0,Y 266.575,Z 367.709,A -85,B 0,C 180,E1 -18108.045,E2 -18108.045} C_VEL
LIN {X 0,Y 268.62,Z 358.619,A -85,B 0,C 180,E1 -18110.282,E2 -18110.282} C_VEL
LIN {X 0,Y 271.116,Z 348.273,A -85,B 0,C 180,E1 -18112.278,E2 -18112.278} C_VEL
LIN {X 0,Y 272.166,Z 342.777,A -85,B 0,C 180,E1 -18113.19,E2 -18113.19} C_VEL
LIN {X 0,Y 272.611,Z 331.214,A -85,B 0,C 180,E1 -18114.985,E2 -18114.985} C_VEL
LIN {X 0,Y 272.163,Z 320.433,A -85,B 0,C 180,E1 -18116.437,E2 -18116.437} C_VEL
LIN {X 0,Y 270.48,Z 308.201,A -85,B 0,C 180,E1 -18117.936,E2 -18117.936} C_VEL
LIN {X 0,Y 267.693,Z 295.992,A -85,B 0,C 180,E1 -18119.326,E2 -18119.326} C_VEL
LIN {X 0,Y 265.134,Z 287.834,A -85,B 0,C 180,E1 -18120.228,E2 -18120.228} C_VEL
LIN {X 0,Y 264.587,Z 285.27,A -85,B 0,C 180,E1 -18120.474,E2 -18120.474} C_VEL
LIN {X 0,Y 266.14,Z 278.602,A -85,B 0,C 180,E1 -18125.517,E2 -18125.517} C_VEL
LIN {X 0,Y 266.488,Z 275.928,A -85,B 0,C 180,E1 -18127.701,E2 -18127.701} C_VEL
LIN {X 0,Y 266.297,Z 273.281,A -85,B 0,C 180,E1 -18130.058,E2 -18130.058} C_VEL
LIN {X 0,Y 265.703,Z 269.808,A -85,B 0,C 180,E1 -18133.448,E2 -18133.448} C_VEL
LIN {X 0,Y 264.975,Z 265.708,A -85,B 0,C 180,E1 -18137.956,E2 -18137.956} C_VEL
LIN {X 0,Y 264.37,Z 262.325,A -85,B 0,C 180,E1 -18142.304,E2 -18142.304} C_VEL
LIN {X 0,Y 263.948,Z 259.88,A -85,B 0,C 180,E1 -18146,E2 -18146} C_VEL
LIN {X 0,Y 263.565,Z 257.966,A -85,B 0,C 180,E1 -18149.557,E2 -18149.557} C_VEL
LIN {X 0,Y 263.338,Z 256.453,A -85,B 0,C 180,E1 -18153.016,E2 -18153.016} C_VEL
LIN {X 0,Y 263.226,Z 255.698,A -85,B 0,C 180,E1 -18155.198,E2 -18155.198} C_VEL
LIN {X 0,Y 263.263,Z 255.686,A -85,B 0,C 180,E1 -18159.691,E2 -18159.691} C_VEL
LIN {X 0,Y 263.35,Z 255.677,A -85,B 0,C 180,E1 -18164.52,E2 -18164.52} C_VEL
LIN {X 0,Y 263.372,Z 255.675,A -85,B 0,C 180,E1 -18169.232,E2 -18169.232} C_VEL
LIN {X 0,Y 263.57,Z 255.654,A -85,B 0,C 180,E1 -18172.336,E2 -18172.336} C_VEL
LIN {X 0,Y 263.749,Z 255.632,A -85,B 0,C 180,E1 -18178.471,E2 -18178.471} C_VEL
LIN {X 0,Y 263.865,Z 256.467,A -85,B 0,C 180,E1 -18181.524,E2 -18181.524} C_VEL
LIN {X 0,Y 263.934,Z 258.552,A -85,B 0,C 180,E1 -18186.88,E2 -18186.88} C_VEL
LIN {X 0,Y 264.025,Z 259.959,A -85,B 0,C 180,E1 -18189.979,E2 -18189.979} C_VEL
LIN {X 0,Y 263.694,Z 262.008,A -85,B 0,C 180,E1 -18193.876,E2 -18193.876} C_VEL
LIN {X 0,Y 263.511,Z 263.612,A -85,B 0,C 180,E1 -18196.523,E2 -18196.523} C_VEL
LIN {X 0,Y 264.689,Z 266.687,A -85,B 0,C 180,E1 -18196.909,E2 -18196.909} C_VEL
LIN {X 0,Y 268.508,Z 274.835,A -85,B 0,C 180,E1 -18198.106,E2 -18198.106} C_VEL
LIN {X 0,Y 272.504,Z 285.79,A -85,B 0,C 180,E1 -18199.713,E2 -18199.713} C_VEL
LIN {X 0,Y 275,Z 295.391,A -85,B 0,C 180,E1 -18201.158,E2 -18201.158} C_VEL
LIN {X 0,Y 276.531,Z 304.235,A -85,B 0,C 180,E1 -18202.569,E2 -18202.569} C_VEL
LIN {X 0,Y 274.522,Z 315.467,A -85,B 0,C 180,E1 -18204.178,E2 -18204.178} C_VEL
LIN {X 0,Y 272.15,Z 325.951,A -85,B 0,C 180,E1 -18206.037,E2 -18206.037} C_VEL
LIN {X 0,Y 270.09,Z 334.392,A -85,B 0,C 180,E1 -18207.926,E2 -18207.926} C_VEL
LIN {X 0,Y 268.01,Z 342.145,A -85,B 0,C 180,E1 -18210.079,E2 -18210.079} C_VEL
LIN {X 0,Y 266.195,Z 348.645,A -85,B 0,C 180,E1 -18212.346,E2 -18212.346} C_VEL
LIN {X 0,Y 264.698,Z 353.769,A -85,B 0,C 180,E1 -18214.608,E2 -18214.608} C_VEL
LIN {X 0,Y 263.538,Z 357.712,A -85,B 0,C 180,E1 -18216.868,E2 -18216.868} C_VEL
LIN {X 0,Y 262.329,Z 361.5,A -85,B 0,C 180,E1 -18220.01,E2 -18220.01} C_VEL
LIN {X 0,Y 261.759,Z 363.074,A -85,B 0,C 180,E1 -18222.158,E2 -18222.158} C_VEL
LIN {X 0,Y 261.382,Z 363.85,A -85,B 0,C 180,E1 -18224.349,E2 -18224.349} C_VEL
LIN {X 0,Y 261.187,Z 363.794,A -85,B 0,C 180,E1 -18226.59,E2 -18226.59} C_VEL
LIN {X 0,Y 261.285,Z 362.258,A -85,B 0,C 180,E1 -18229.795,E2 -18229.795} C_VEL
LIN {X 0,Y 261.761,Z 359.224,A -85,B 0,C 180,E1 -18232.778,E2 -18232.778} C_VEL
LIN {X 0,Y 262.522,Z 354.427,A -85,B 0,C 180,E1 -18235.794,E2 -18235.794} C_VEL
LIN {X 0,Y 263.537,Z 348.297,A -85,B 0,C 180,E1 -18238.574,E2 -18238.574} C_VEL
LIN {X 0,Y 264.855,Z 340.894,A -85,B 0,C 180,E1 -18241.117,E2 -18241.117} C_VEL
LIN {X 0,Y 266.25,Z 332.757,A -85,B 0,C 180,E1 -18243.338,E2 -18243.338} C_VEL
LIN {X 0,Y 267.661,Z 324.55,A -85,B 0,C 180,E1 -18245.159,E2 -18245.159} C_VEL
LIN {X 0,Y 269.24,Z 314.652,A -85,B 0,C 180,E1 -18246.95,E2 -18246.95} C_VEL
LIN {X 0,Y 270.806,Z 303.991,A -85,B 0,C 180,E1 -18248.496,E2 -18248.496} C_VEL
LIN {X 0,Y 271.604,Z 297.45,A -85,B 0,C 180,E1 -18249.298,E2 -18249.298} C_VEL
LIN {X 0,Y 269.682,Z 287.101,A -85,B 0,C 180,E1 -18250.594,E2 -18250.594} C_VEL
LIN {X 0,Y 266.655,Z 274.568,A -85,B 0,C 180,E1 -18251.921,E2 -18251.921} C_VEL
LIN {X 0,Y 262.884,Z 261.781,A -85,B 0,C 180,E1 -18253.024,E2 -18253.024} C_VEL
LIN {X 0,Y 262.315,Z 259.513,A -85,B 0,C 180,E1 -18253.212,E2 -18253.212} C_VEL
LIN {X 0,Y 262.597,Z 256.056,A -85,B 0,C 180,E1 -18257.638,E2 -18257.638} C_VEL
LIN {X 0,Y 263.208,Z 255.699,A -85,B 0,C 180,E1 -18261.073,E2 -18261.073} C_VEL
LIN {X 0,Y 263.442,Z 255.671,A -85,B 0,C 180,E1 -18263.875,E2 -18263.875} C_VEL
LIN {X 0,Y 263.741,Z 255.632,A -85,B 0,C 180,E1 -18268.474,E2 -18268.474} C_VEL
LIN {X 0,Y 263.738,Z 255.633,A -85,B 0,C 180,E1 -18271.528,E2 -18271.528} C_VEL
LIN {X 0,Y 263.558,Z 255.654,A -85,B 0,C 180,E1 -18277.663,E2 -18277.663} C_VEL
LIN {X 0,Y 263.361,Z 255.68,A -85,B 0,C 180,E1 -18280.767,E2 -18280.767} C_VEL
LIN {X 0,Y 263.338,Z 255.683,A -85,B 0,C 180,E1 -18285.48,E2 -18285.48} C_VEL
LIN {X 0,Y 263.28,Z 255.688,A -85,B 0,C 180,E1 -18290.306,E2 -18290.306} C_VEL
LIN {X 0,Y 263.226,Z 255.698,A -85,B 0,C 180,E1 -18294.807,E2 -18294.807} C_VEL
LIN {X 0,Y 263.169,Z 255.704,A -85,B 0,C 180,E1 -18298.732,E2 -18298.732} C_VEL
LIN {X 0,Y 263.123,Z 255.71,A -85,B 0,C 180,E1 -18302.29,E2 -18302.29} C_VEL
LIN {X 0,Y 263.178,Z 255.697,A -85,B 0,C 180,E1 -18305.98,E2 -18305.98} C_VEL
LIN {X 0,Y 263.153,Z 255.703,A -85,B 0,C 180,E1 -18309.865,E2 -18309.865} C_VEL
LIN {X 0,Y 263.184,Z 255.699,A -85,B 0,C 180,E1 -18313.867,E2 -18313.867} C_VEL
LIN {X 0,Y 263.206,Z 255.694,A -85,B 0,C 180,E1 -18318.388,E2 -18318.388} C_VEL
LIN {X 0,Y 263.201,Z 255.697,A -85,B 0,C 180,E1 -18323.233,E2 -18323.233} C_VEL
LIN {X 0,Y 263.179,Z 255.701,A -85,B 0,C 180,E1 -18325.893,E2 -18325.893} C_VEL
LIN {X 0,Y 263.144,Z 255.698,A -85,B 0,C 180,E1 -18329.51,E2 -18329.51} C_VEL
LIN {X 0,Y 263.189,Z 255.697,A -85,B 0,C 180,E1 -18333.006,E2 -18333.006} C_VEL
LIN {X 0,Y 263.182,Z 255.702,A -85,B 0,C 180,E1 -18336.39,E2 -18336.39} C_VEL
LIN {X 0,Y 263.262,Z 255.689,A -85,B 0,C 180,E1 -18339.696,E2 -18339.696} C_VEL
LIN {X 0,Y 263.351,Z 255.676,A -85,B 0,C 180,E1 -18344.525,E2 -18344.525} C_VEL
LIN {X 0,Y 263.355,Z 255.678,A -85,B 0,C 180,E1 -18349.236,E2 -18349.236} C_VEL
LIN {X 0,Y 263.546,Z 255.653,A -85,B 0,C 180,E1 -18352.34,E2 -18352.34} C_VEL
LIN {X 0,Y 263.754,Z 255.627,A -85,B 0,C 180,E1 -18358.476,E2 -18358.476} C_VEL
LIN {X 0,Y 263.753,Z 255.631,A -85,B 0,C 180,E1 -18361.529,E2 -18361.529} C_VEL
LIN {X 0,Y 263.536,Z 255.654,A -85,B 0,C 180,E1 -18367.665,E2 -18367.665} C_VEL
LIN {X 0,Y 263.355,Z 255.678,A -85,B 0,C 180,E1 -18370.769,E2 -18370.769} C_VEL
LIN {X 0,Y 263.357,Z 255.678,A -85,B 0,C 180,E1 -18375.48,E2 -18375.48} C_VEL
LIN {X 0,Y 263.27,Z 255.689,A -85,B 0,C 180,E1 -18380.308,E2 -18380.308} C_VEL
LIN {X 0,Y 263.215,Z 255.7,A -85,B 0,C 180,E1 -18385.293,E2 -18385.293} C_VEL
LIN {X 0,Y 263.178,Z 255.7,A -85,B 0,C 180,E1 -18386.078,E2 -18386.078} C_VEL
LIN {X 0,Y 262.493,Z 255.79,A -85,B 0,C 180,E1 -18387.354,E2 -18387.354} C_VEL
LIN {X 0,Y 259.6,Z 256.15,A -85,B 0,C 180,E1 -18389.433,E2 -18389.433} C_VEL
LIN {X 0,Y 257.162,Z 256.453,A -85,B 0,C 180,E1 -18391.124,E2 -18391.124} C_VEL
LIN {X 0,Y 256.134,Z 256.579,A -85,B 0,C 180,E1 -18392.436,E2 -18392.436} C_VEL
LIN {X 0,Y 256.06,Z 256.588,A -85,B 0,C 180,E1 -18392.881,E2 -18392.881} C_VEL
LIN {X 0,Y 256.154,Z 256.579,A -85,B 0,C 180,E1 -18397.131,E2 -18397.131} C_VEL
LIN {X 0,Y 256.163,Z 256.635,A -85,B 0,C 180,E1 -18397.634,E2 -18397.634} C_VEL
LIN {X 0,Y 257.042,Z 261.709,A -85,B 0,C 180,E1 -18402.418,E2 -18402.418} C_VEL
LIN {X 0,Y 258.076,Z 267.268,A -85,B 0,C 180,E1 -18407.333,E2 -18407.333} C_VEL
LIN {X 0,Y 258.908,Z 272.197,A -85,B 0,C 180,E1 -18411.366,E2 -18411.366} C_VEL
LIN {X 0,Y 258.884,Z 274.717,A -85,B 0,C 180,E1 -18413.327,E2 -18413.327} C_VEL
LIN {X 0,Y 258.19,Z 278.451,A -85,B 0,C 180,E1 -18416.08,E2 -18416.08} C_VEL
LIN {X 0,Y 257.004,Z 284.594,A -85,B 0,C 180,E1 -18420.512,E2 -18420.512} C_VEL
LIN {X 0,Y 256.439,Z 287.86,A -85,B 0,C 180,E1 -18422.839,E2 -18422.839} C_VEL
LIN {X 0,Y 258.843,Z 301.403,A -85,B 0,C 180,E1 -18423.784,E2 -18423.784} C_VEL
LIN {X 0,Y 260.689,Z 314.769,A -85,B 0,C 180,E1 -18425.013,E2 -18425.013} C_VEL
LIN {X 0,Y 261.833,Z 327.148,A -85,B 0,C 180,E1 -18426.425,E2 -18426.425} C_VEL
LIN {X 0,Y 262.369,Z 338.292,A -85,B 0,C 180,E1 -18427.974,E2 -18427.974} C_VEL
LIN {X 0,Y 262.132,Z 342.2,A -85,B 0,C 180,E1 -18428.573,E2 -18428.573} C_VEL
LIN {X 0,Y 260.338,Z 352.137,A -85,B 0,C 180,E1 -18430.278,E2 -18430.278} C_VEL
LIN {X 0,Y 258.684,Z 361.628,A -85,B 0,C 180,E1 -18432.31,E2 -18432.31} C_VEL
LIN {X 0,Y 257.134,Z 370.045,A -85,B 0,C 180,E1 -18434.544,E2 -18434.544} C_VEL
LIN {X 0,Y 255.853,Z 377.136,A -85,B 0,C 180,E1 -18436.901,E2 -18436.901} C_VEL
LIN {X 0,Y 254.9,Z 383.606,A -85,B 0,C 180,E1 -18439.675,E2 -18439.675} C_VEL
LIN {X 0,Y 254.421,Z 387.855,A -85,B 0,C 180,E1 -18442.06,E2 -18442.06} C_VEL
LIN {X 0,Y 254.26,Z 390.885,A -85,B 0,C 180,E1 -18444.329,E2 -18444.329} C_VEL
LIN {X 0,Y 254.215,Z 393.169,A -85,B 0,C 180,E1 -18446.83,E2 -18446.83} C_VEL
LIN {X 0,Y 254.184,Z 394.071,A -85,B 0,C 180,E1 -18448.415,E2 -18448.415} C_VEL
LIN {X 0,Y 254.259,Z 394.575,A -85,B 0,C 180,E1 -18449.999,E2 -18449.999} C_VEL
LIN {X 0,Y 254.178,Z 394.625,A -85,B 0,C 180,E1 -18451.584,E2 -18451.584} C_VEL
LIN {X 0,Y 254.172,Z 394.273,A -85,B 0,C 180,E1 -18453.169,E2 -18453.169} C_VEL
LIN {X 0,Y 254.237,Z 392.39,A -85,B 0,C 180,E1 -18456.347,E2 -18456.347} C_VEL
LIN {X 0,Y 254.513,Z 389.87,A -85,B 0,C 180,E1 -18458.735,E2 -18458.735} C_VEL
LIN {X 0,Y 255.123,Z 386.376,A -85,B 0,C 180,E1 -18461.117,E2 -18461.117} C_VEL
LIN {X 0,Y 256.114,Z 381.833,A -85,B 0,C 180,E1 -18463.487,E2 -18463.487} C_VEL
LIN {X 0,Y 257.94,Z 375.069,A -85,B 0,C 180,E1 -18466.216,E2 -18466.216} C_VEL
LIN {X 0,Y 259.881,Z 367.447,A -85,B 0,C 180,E1 -18468.623,E2 -18468.623} C_VEL
LIN {X 0,Y 261.979,Z 358.81,A -85,B 0,C 180,E1 -18470.82,E2 -18470.82} C_VEL
LIN {X 0,Y 264.583,Z 348.657,A -85,B 0,C 180,E1 -18472.859,E2 -18472.859} C_VEL
LIN {X 0,Y 265.616,Z 343.245,A -85,B 0,C 180,E1 -18473.796,E2 -18473.796} C_VEL
LIN {X 0,Y 266.152,Z 332.152,A -85,B 0,C 180,E1 -18475.595,E2 -18475.595} C_VEL
LIN {X 0,Y 265.812,Z 321.411,A -85,B 0,C 180,E1 -18477.137,E2 -18477.137} C_VEL
LIN {X 0,Y 264.337,Z 309.745,A -85,B 0,C 180,E1 -18478.668,E2 -18478.668} C_VEL
LIN {X 0,Y 261.534,Z 297.136,A -85,B 0,C 180,E1 -18480.199,E2 -18480.199} C_VEL
LIN {X 0,Y 258.712,Z 288.062,A -85,B 0,C 180,E1 -18481.293,E2 -18481.293} C_VEL
LIN {X 0,Y 257.853,Z 284.733,A -85,B 0,C 180,E1 -18481.645,E2 -18481.645} C_VEL
LIN {X 0,Y 259.089,Z 279.785,A -85,B 0,C 180,E1 -18485.53,E2 -18485.53} C_VEL
LIN {X 0,Y 259.456,Z 276.6,A -85,B 0,C 180,E1 -18488.227,E2 -18488.227} C_VEL
LIN {X 0,Y 259.21,Z 274.05,A -85,B 0,C 180,E1 -18490.606,E2 -18490.606} C_VEL
LIN {X 0,Y 258.845,Z 271.814,A -85,B 0,C 180,E1 -18492.851,E2 -18492.851} C_VEL
LIN {X 0,Y 258.1,Z 267.785,A -85,B 0,C 180,E1 -18497.323,E2 -18497.323} C_VEL
LIN {X 0,Y 257.581,Z 264.803,A -85,B 0,C 180,E1 -18501.128,E2 -18501.128} C_VEL
LIN {X 0,Y 257.121,Z 262.215,A -85,B 0,C 180,E1 -18504.968,E2 -18504.968} C_VEL
LIN {X 0,Y 256.734,Z 260.13,A -85,B 0,C 180,E1 -18508.657,E2 -18508.657} C_VEL
LIN {X 0,Y 256.476,Z 258.507,A -85,B 0,C 180,E1 -18512.233,E2 -18512.233} C_VEL
LIN {X 0,Y 256.3,Z 257.278,A -85,B 0,C 180,E1 -18515.71,E2 -18515.71} C_VEL
LIN {X 0,Y 256.167,Z 256.573,A -85,B 0,C 180,E1 -18519.102,E2 -18519.102} C_VEL
LIN {X 0,Y 256.299,Z 256.556,A -85,B 0,C 180,E1 -18524.083,E2 -18524.083} C_VEL
LIN {X 0,Y 256.308,Z 256.555,A -85,B 0,C 180,E1 -18528.931,E2 -18528.931} C_VEL
LIN {X 0,Y 256.538,Z 256.528,A -85,B 0,C 180,E1 -18532.124,E2 -18532.124} C_VEL
LIN {X 0,Y 256.53,Z 256.75,A -85,B 0,C 180,E1 -18536.856,E2 -18536.856} C_VEL
LIN {X 0,Y 256.949,Z 257.497,A -85,B 0,C 180,E1 -18539.997,E2 -18539.997} C_VEL
LIN {X 0,Y 256.845,Z 258.554,A -85,B 0,C 180,E1 -18543.134,E2 -18543.134} C_VEL
LIN {X 0,Y 257.05,Z 260.373,A -85,B 0,C 180,E1 -18547.854,E2 -18547.854} C_VEL
LIN {X 0,Y 257.032,Z 261.415,A -85,B 0,C 180,E1 -18550.158,E2 -18550.158} C_VEL
LIN {X 0,Y 256.68,Z 263.505,A -85,B 0,C 180,E1 -18554.263,E2 -18554.263} C_VEL
LIN {X 0,Y 256.607,Z 264.065,A -85,B 0,C 180,E1 -18555.281,E2 -18555.281} C_VEL
LIN {X 0,Y 257.775,Z 267.187,A -85,B 0,C 180,E1 -18555.717,E2 -18555.717} C_VEL
LIN {X 0,Y 259.018,Z 269.558,A -85,B 0,C 180,E1 -18556.103,E2 -18556.103} C_VEL
LIN {X 0,Y 263.304,Z 279.128,A -85,B 0,C 180,E1 -18557.622,E2 -18557.622} C_VEL
LIN {X 0,Y 266.589,Z 288.734,A -85,B 0,C 180,E1 -18559.137,E2 -18559.137} C_VEL
LIN {X 0,Y 268.986,Z 298.53,A -85,B 0,C 180,E1 -18560.716,E2 -18560.716} C_VEL
LIN {X 0,Y 270.198,Z 305.801,A -85,B 0,C 180,E1 -18561.953,E2 -18561.953} C_VEL
LIN {X 0,Y 268.234,Z 316.235,A -85,B 0,C 180,E1 -18563.507,E2 -18563.507} C_VEL
LIN {X 0,Y 265.769,Z 326.467,A -85,B 0,C 180,E1 -18565.37,E2 -18565.37} C_VEL
LIN {X 0,Y 263.417,Z 335.573,A -85,B 0,C 180,E1 -18567.478,E2 -18567.478} C_VEL
LIN {X 0,Y 261.289,Z 343.012,A -85,B 0,C 180,E1 -18569.618,E2 -18569.618} C_VEL
LIN {X 0,Y 259.183,Z 350.155,A -85,B 0,C 180,E1 -18572.23,E2 -18572.23} C_VEL
LIN {X 0,Y 257.402,Z 355.83,A -85,B 0,C 180,E1 -18575.006,E2 -18575.006} C_VEL
LIN {X 0,Y 256.253,Z 359.348,A -85,B 0,C 180,E1 -18577.313,E2 -18577.313} C_VEL
LIN {X 0,Y 255.37,Z 361.873,A -85,B 0,C 180,E1 -18579.595,E2 -18579.595} C_VEL
LIN {X 0,Y 254.739,Z 363.504,A -85,B 0,C 180,E1 -18581.851,E2 -18581.851} C_VEL
LIN {X 0,Y 254.333,Z 364.279,A -85,B 0,C 180,E1 -18584.074,E2 -18584.074} C_VEL
LIN {X 0,Y 254.146,Z 364.265,A -85,B 0,C 180,E1 -18586.266,E2 -18586.266} C_VEL
LIN {X 0,Y 254.099,Z 363.53,A -85,B 0,C 180,E1 -18588.411,E2 -18588.411} C_VEL
LIN {X 0,Y 254.326,Z 361.942,A -85,B 0,C 180,E1 -18590.686,E2 -18590.686} C_VEL
LIN {X 0,Y 254.756,Z 359.258,A -85,B 0,C 180,E1 -18593.127,E2 -18593.127} C_VEL
LIN {X 0,Y 255.368,Z 355.348,A -85,B 0,C 180,E1 -18595.647,E2 -18595.647} C_VEL
LIN {X 0,Y 256.299,Z 350.039,A -85,B 0,C 180,E1 -18598.211,E2 -18598.211} C_VEL
LIN {X 0,Y 257.545,Z 343.051,A -85,B 0,C 180,E1 -18600.829,E2 -18600.829} C_VEL
LIN {X 0,Y 258.906,Z 335.604,A -85,B 0,C 180,E1 -18603.037,E2 -18603.037} C_VEL
LIN {X 0,Y 260.636,Z 326.048,A -85,B 0,C 180,E1 -18605.296,E2 -18605.296} C_VEL
LIN {X 0,Y 262.216,Z 316.447,A -85,B 0,C 180,E1 -18607.132,E2 -18607.132} C_VEL
LIN {X 0,Y 263.866,Z 305.724,A -85,B 0,C 180,E1 -18608.774,E2 -18608.774} C_VEL
LIN {X 0,Y 264.705,Z 297.657,A -85,B 0,C 180,E1 -18609.81,E2 -18609.81} C_VEL
LIN {X 0,Y 262.469,Z 286.347,A -85,B 0,C 180,E1 -18611.258,E2 -18611.258} C_VEL
LIN {X 0,Y 259.221,Z 273.26,A -85,B 0,C 180,E1 -18612.65,E2 -18612.65} C_VEL
LIN {X 0,Y 255.285,Z 259.911,A -85,B 0,C 180,E1 -18613.836,E2 -18613.836} C_VEL
LIN {X 0,Y 255.519,Z 257.27,A -85,B 0,C 180,E1 -18617.29,E2 -18617.29} C_VEL
LIN {X 0,Y 255.708,Z 256.635,A -85,B 0,C 180,E1 -18618.909,E2 -18618.909} C_VEL
LIN {X 0,Y 256.299,Z 256.559,A -85,B 0,C 180,E1 -18622.121,E2 -18622.121} C_VEL
LIN {X 0,Y 256.309,Z 256.562,A -85,B 0,C 180,E1 -18625.282,E2 -18625.282} C_VEL
LIN {X 0,Y 256.703,Z 256.509,A -85,B 0,C 180,E1 -18628.432,E2 -18628.432} C_VEL
LIN {X 0,Y 256.701,Z 256.509,A -85,B 0,C 180,E1 -18631.57,E2 -18631.57} C_VEL
LIN {X 0,Y 256.526,Z 256.529,A -85,B 0,C 180,E1 -18637.874,E2 -18637.874} C_VEL
LIN {X 0,Y 256.297,Z 256.56,A -85,B 0,C 180,E1 -18641.067,E2 -18641.067} C_VEL
LIN {X 0,Y 256.287,Z 256.561,A -85,B 0,C 180,E1 -18645.917,E2 -18645.917} C_VEL
LIN {X 0,Y 256.229,Z 256.571,A -85,B 0,C 180,E1 -18650.891,E2 -18650.891} C_VEL
LIN {X 0,Y 256.186,Z 256.572,A -85,B 0,C 180,E1 -18655.145,E2 -18655.145} C_VEL
LIN {X 0,Y 256.103,Z 256.582,A -85,B 0,C 180,E1 -18659.602,E2 -18659.602} C_VEL
LIN {X 0,Y 256.075,Z 256.585,A -85,B 0,C 180,E1 -18663.293,E2 -18663.293} C_VEL
LIN {X 0,Y 256.13,Z 256.575,A -85,B 0,C 180,E1 -18667.281,E2 -18667.281} C_VEL
LIN {X 0,Y 256.125,Z 256.58,A -85,B 0,C 180,E1 -18671.191,E2 -18671.191} C_VEL
LIN {X 0,Y 256.109,Z 256.577,A -85,B 0,C 180,E1 -18675.519,E2 -18675.519} C_VEL
LIN {X 0,Y 256.126,Z 256.577,A -85,B 0,C 180,E1 -18678.815,E2 -18678.815} C_VEL
LIN {X 0,Y 256.15,Z 256.577,A -85,B 0,C 180,E1 -18682.875,E2 -18682.875} C_VEL
LIN {X 0,Y 256.081,Z 256.583,A -85,B 0,C 180,E1 -18686.713,E2 -18686.713} C_VEL
LIN {X 0,Y 256.131,Z 256.572,A -85,B 0,C 180,E1 -18691.409,E2 -18691.409} C_VEL
LIN {X 0,Y 256.165,Z 256.574,A -85,B 0,C 180,E1 -18695.702,E2 -18695.702} C_VEL
LIN {X 0,Y 256.165,Z 256.572,A -85,B 0,C 180,E1 -18699.108,E2 -18699.108} C_VEL
LIN {X 0,Y 256.3,Z 256.554,A -85,B 0,C 180,E1 -18704.088,E2 -18704.088} C_VEL
LIN {X 0,Y 256.298,Z 256.557,A -85,B 0,C 180,E1 -18708.936,E2 -18708.936} C_VEL
LIN {X 0,Y 256.506,Z 256.531,A -85,B 0,C 180,E1 -18712.129,E2 -18712.129} C_VEL
LIN {X 0,Y 256.499,Z 256.527,A -85,B 0,C 180,E1 -18716.861,E2 -18716.861} C_VEL
LIN {X 0,Y 256.768,Z 256.501,A -85,B 0,C 180,E1 -18720.003,E2 -18720.003} C_VEL
LIN {X 0,Y 256.497,Z 256.533,A -85,B 0,C 180,E1 -18723.144,E2 -18723.144} C_VEL
LIN {X 0,Y 256.499,Z 256.532,A -85,B 0,C 180,E1 -18727.877,E2 -18727.877} C_VEL
LIN {X 0,Y 256.297,Z 256.558,A -85,B 0,C 180,E1 -18731.069,E2 -18731.069} C_VEL
LIN {X 0,Y 256.306,Z 256.554,A -85,B 0,C 180,E1 -18735.917,E2 -18735.917} C_VEL
LIN {X 0,Y 256.174,Z 256.574,A -85,B 0,C 180,E1 -18740.897,E2 -18740.897} C_VEL
LIN {X 0,Y 256.195,Z 256.573,A -85,B 0,C 180,E1 -18745.14,E2 -18745.14} C_VEL
LIN {X 0,Y 256.111,Z 256.583,A -85,B 0,C 180,E1 -18749.603,E2 -18749.603} C_VEL
LIN {X 0,Y 256.06,Z 256.588,A -85,B 0,C 180,E1 -18752.881,E2 -18752.881} C_VEL
LIN {X 0,Y 255.375,Z 256.706,A -85,B 0,C 180,E1 -18753.762,E2 -18753.762} C_VEL
LIN {X 0,Y 252.475,Z 257.037,A -85,B 0,C 180,E1 -18755.146,E2 -18755.146} C_VEL
LIN {X 0,Y 249.678,Z 257.385,A -85,B 0,C 180,E1 -18756.55,E2 -18756.55} C_VEL
LIN {X 0,Y 249.161,Z 257.785,A -85,B 0,C 180,E1 -18757.445,E2 -18757.445} C_VEL
LIN {X 0,Y 250.06,Z 262.911,A -85,B 0,C 180,E1 -18762.42,E2 -18762.42} C_VEL
LIN {X 0,Y 250.928,Z 267.695,A -85,B 0,C 180,E1 -18766.739,E2 -18766.739} C_VEL
LIN {X 0,Y 251.639,Z 271.513,A -85,B 0,C 180,E1 -18770.031,E2 -18770.031} C_VEL
LIN {X 0,Y 251.87,Z 274.074,A -85,B 0,C 180,E1 -18772.129,E2 -18772.129} C_VEL
LIN {X 0,Y 251.679,Z 276.607,A -85,B 0,C 180,E1 -18774.096,E2 -18774.096} C_VEL
LIN {X 0,Y 250.387,Z 282.747,A -85,B 0,C 180,E1 -18778.716,E2 -18778.716} C_VEL
LIN {X 0,Y 249.529,Z 287.489,A -85,B 0,C 180,E1 -18782.194,E2 -18782.194} C_VEL
LIN {X 0,Y 251.88,Z 300.999,A -85,B 0,C 180,E1 -18783.17,E2 -18783.17} C_VEL
LIN {X 0,Y 253.559,Z 313.278,A -85,B 0,C 180,E1 -18784.325,E2 -18784.325} C_VEL
LIN {X 0,Y 254.748,Z 325.756,A -85,B 0,C 180,E1 -18785.775,E2 -18785.775} C_VEL
LIN {X 0,Y 255.368,Z 336.832,A -85,B 0,C 180,E1 -18787.337,E2 -18787.337} C_VEL
LIN {X 0,Y 255.276,Z 342.133,A -85,B 0,C 180,E1 -18788.181,E2 -18788.181} C_VEL
LIN {X 0,Y 253.595,Z 351.009,A -85,B 0,C 180,E1 -18789.731,E2 -18789.731} C_VEL
LIN {X 0,Y 251.864,Z 360.345,A -85,B 0,C 180,E1 -18791.746,E2 -18791.746} C_VEL
LIN {X 0,Y 250.493,Z 367.775,A -85,B 0,C 180,E1 -18793.705,E2 -18793.705} C_VEL
LIN {X 0,Y 249.106,Z 375.221,A -85,B 0,C 180,E1 -18796.124,E2 -18796.124} C_VEL
LIN {X 0,Y 248.113,Z 381.197,A -85,B 0,C 180,E1 -18798.563,E2 -18798.563} C_VEL
LIN {X 0,Y 247.516,Z 385.909,A -85,B 0,C 180,E1 -18801.015,E2 -18801.015} C_VEL
LIN {X 0,Y 247.197,Z 389.481,A -85,B 0,C 180,E1 -18803.469,E2 -18803.469} C_VEL
LIN {X 0,Y 247.134,Z 391.298,A -85,B 0,C 180,E1 -18805.105,E2 -18805.105} C_VEL
LIN {X 0,Y 247.149,Z 392.643,A -85,B 0,C 180,E1 -18806.739,E2 -18806.739} C_VEL
LIN {X 0,Y 247.111,Z 393.572,A -85,B 0,C 180,E1 -18808.369,E2 -18808.369} C_VEL
LIN {X 0,Y 247.179,Z 394.105,A -85,B 0,C 180,E1 -18809.999,E2 -18809.999} C_VEL
LIN {X 0,Y 247.104,Z 394.208,A -85,B 0,C 180,E1 -18811.629,E2 -18811.629} C_VEL
LIN {X 0,Y 247.083,Z 393.881,A -85,B 0,C 180,E1 -18813.26,E2 -18813.26} C_VEL
LIN {X 0,Y 247.169,Z 392.05,A -85,B 0,C 180,E1 -18816.53,E2 -18816.53} C_VEL
LIN {X 0,Y 247.338,Z 390.528,A -85,B 0,C 180,E1 -18818.167,E2 -18818.167} C_VEL
LIN {X 0,Y 248.131,Z 386.161,A -85,B 0,C 180,E1 -18821.435,E2 -18821.435} C_VEL
LIN {X 0,Y 249.184,Z 381.702,A -85,B 0,C 180,E1 -18823.87,E2 -18823.87} C_VEL
LIN {X 0,Y 251.103,Z 375.061,A -85,B 0,C 180,E1 -18826.67,E2 -18826.67} C_VEL
LIN {X 0,Y 253.029,Z 368.012,A -85,B 0,C 180,E1 -18828.999,E2 -18828.999} C_VEL
LIN {X 0,Y 255.351,Z 359.001,A -85,B 0,C 180,E1 -18831.387,E2 -18831.387} C_VEL
LIN {X 0,Y 258.08,Z 349.04,A -85,B 0,C 180,E1 -18833.469,E2 -18833.469} C_VEL
LIN {X 0,Y 259.092,Z 343.755,A -85,B 0,C 180,E1 -18834.434,E2 -18834.434} C_VEL
LIN {X 0,Y 259.797,Z 331.436,A -85,B 0,C 180,E1 -18836.516,E2 -18836.516} C_VEL
LIN {X 0,Y 259.383,Z 320.75,A -85,B 0,C 180,E1 -18838.113,E2 -18838.113} C_VEL
LIN {X 0,Y 257.789,Z 308.835,A -85,B 0,C 180,E1 -18839.754,E2 -18839.754} C_VEL
LIN {X 0,Y 254.96,Z 296.419,A -85,B 0,C 180,E1 -18841.373,E2 -18841.373} C_VEL
LIN {X 0,Y 252.048,Z 287.548,A -85,B 0,C 180,E1 -18842.531,E2 -18842.531} C_VEL
LIN {X 0,Y 251.194,Z 284.164,A -85,B 0,C 180,E1 -18842.925,E2 -18842.925} C_VEL
LIN {X 0,Y 252.209,Z 280.329,A -85,B 0,C 180,E1 -18846.085,E2 -18846.085} C_VEL
LIN {X 0,Y 252.437,Z 277.294,A -85,B 0,C 180,E1 -18848.779,E2 -18848.779} C_VEL
LIN {X 0,Y 252.042,Z 274.028,A -85,B 0,C 180,E1 -18852.005,E2 -18852.005} C_VEL
LIN {X 0,Y 251.243,Z 269.871,A -85,B 0,C 180,E1 -18856.659,E2 -18856.659} C_VEL
LIN {X 0,Y 250.839,Z 267.313,A -85,B 0,C 180,E1 -18859.875,E2 -18859.875} C_VEL
LIN {X 0,Y 250.348,Z 264.556,A -85,B 0,C 180,E1 -18863.874,E2 -18863.874} C_VEL
LIN {X 0,Y 249.961,Z 262.339,A -85,B 0,C 180,E1 -18867.707,E2 -18867.707} C_VEL
LIN {X 0,Y 249.651,Z 260.596,A -85,B 0,C 180,E1 -18871.405,E2 -18871.405} C_VEL
LIN {X 0,Y 249.482,Z 259.241,A -85,B 0,C 180,E1 -18875.001,E2 -18875.001} C_VEL
LIN {X 0,Y 249.199,Z 257.967,A -85,B 0,C 180,E1 -18880.216,E2 -18880.216} C_VEL
LIN {X 0,Y 249.241,Z 257.491,A -85,B 0,C 180,E1 -18883.619,E2 -18883.619} C_VEL
LIN {X 0,Y 249.251,Z 257.435,A -85,B 0,C 180,E1 -18888.614,E2 -18888.614} C_VEL
LIN {X 0,Y 249.503,Z 257.541,A -85,B 0,C 180,E1 -18891.901,E2 -18891.901} C_VEL
LIN {X 0,Y 249.616,Z 258.33,A -85,B 0,C 180,E1 -18896.769,E2 -18896.769} C_VEL
LIN {X 0,Y 250.041,Z 259.043,A -85,B 0,C 180,E1 -18899.997,E2 -18899.997} C_VEL
LIN {X 0,Y 249.91,Z 260.078,A -85,B 0,C 180,E1 -18903.222,E2 -18903.222} C_VEL
LIN {X 0,Y 250.024,Z 261.418,A -85,B 0,C 180,E1 -18906.9,E2 -18906.9} C_VEL
LIN {X 0,Y 250.044,Z 262.891,A -85,B 0,C 180,E1 -18910.35,E2 -18910.35} C_VEL
LIN {X 0,Y 249.747,Z 264.802,A -85,B 0,C 180,E1 -18913.992,E2 -18913.992} C_VEL
LIN {X 0,Y 250.941,Z 267.866,A -85,B 0,C 180,E1 -18914.441,E2 -18914.441} C_VEL
LIN {X 0,Y 252.053,Z 269.696,A -85,B 0,C 180,E1 -18914.789,E2 -18914.789} C_VEL
LIN {X 0,Y 256.709,Z 279.957,A -85,B 0,C 180,E1 -18916.55,E2 -18916.55} C_VEL
LIN {X 0,Y 260.191,Z 289.874,A -85,B 0,C 180,E1 -18918.226,E2 -18918.226} C_VEL
LIN {X 0,Y 262.65,Z 299.863,A -85,B 0,C 180,E1 -18919.945,E2 -18919.945} C_VEL
LIN {X 0,Y 263.877,Z 308.475,A -85,B 0,C 180,E1 -18921.487,E2 -18921.487} C_VEL
LIN {X 0,Y 261.608,Z 318.72,A -85,B 0,C 180,E1 -18923.079,E2 -18923.079} C_VEL
LIN {X 0,Y 258.941,Z 328.972,A -85,B 0,C 180,E1 -18925.089,E2 -18925.089} C_VEL
LIN {X 0,Y 256.416,Z 337.988,A -85,B 0,C 180,E1 -18927.325,E2 -18927.325} C_VEL
LIN {X 0,Y 254.339,Z 344.803,A -85,B 0,C 180,E1 -18929.438,E2 -18929.438} C_VEL
LIN {X 0,Y 252.272,Z 351.238,A -85,B 0,C 180,E1 -18931.956,E2 -18931.956} C_VEL
LIN {X 0,Y 250.477,Z 356.659,A -85,B 0,C 180,E1 -18934.74,E2 -18934.74} C_VEL
LIN {X 0,Y 249.663,Z 358.957,A -85,B 0,C 180,E1 -18936.235,E2 -18936.235} C_VEL
LIN {X 0,Y 248.718,Z 361.564,A -85,B 0,C 180,E1 -18938.433,E2 -18938.433} C_VEL
LIN {X 0,Y 247.956,Z 363.423,A -85,B 0,C 180,E1 -18940.681,E2 -18940.681} C_VEL
LIN {X 0,Y 247.423,Z 364.521,A -85,B 0,C 180,E1 -18942.973,E2 -18942.973} C_VEL
LIN {X 0,Y 247.112,Z 364.821,A -85,B 0,C 180,E1 -18945.313,E2 -18945.313} C_VEL
LIN {X 0,Y 246.996,Z 364.252,A -85,B 0,C 180,E1 -18947.709,E2 -18947.709} C_VEL
LIN {X 0,Y 247.153,Z 362.781,A -85,B 0,C 180,E1 -18950.149,E2 -18950.149} C_VEL
LIN {X 0,Y 247.718,Z 359.324,A -85,B 0,C 180,E1 -18953.432,E2 -18953.432} C_VEL
LIN {X 0,Y 248.244,Z 356.201,A -85,B 0,C 180,E1 -18955.514,E2 -18955.514} C_VEL
LIN {X 0,Y 249.045,Z 351.719,A -85,B 0,C 180,E1 -18957.837,E2 -18957.837} C_VEL
LIN {X 0,Y 250.247,Z 345.054,A -85,B 0,C 180,E1 -18960.523,E2 -18960.523} C_VEL
LIN {X 0,Y 251.687,Z 337.567,A -85,B 0,C 180,E1 -18962.906,E2 -18962.906} C_VEL
LIN {X 0,Y 253.35,Z 328.615,A -85,B 0,C 180,E1 -18965.194,E2 -18965.194} C_VEL
LIN {X 0,Y 255.181,Z 318.094,A -85,B 0,C 180,E1 -18967.321,E2 -18967.321} C_VEL
LIN {X 0,Y 256.809,Z 308.238,A -85,B 0,C 180,E1 -18968.924,E2 -18968.924} C_VEL
LIN {X 0,Y 257.976,Z 299.558,A -85,B 0,C 180,E1 -18970.092,E2 -18970.092} C_VEL
LIN {X 0,Y 255.853,Z 288.369,A -85,B 0,C 180,E1 -18971.606,E2 -18971.606} C_VEL
LIN {X 0,Y 252.832,Z 275.757,A -85,B 0,C 180,E1 -18973.037,E2 -18973.037} C_VEL
LIN {X 0,Y 248.85,Z 262.499,A -85,B 0,C 180,E1 -18974.283,E2 -18974.283} C_VEL
LIN {X 0,Y 248.287,Z 260.324,A -85,B 0,C 180,E1 -18974.476,E2 -18974.476} C_VEL
LIN {X 0,Y 248.597,Z 257.521,A -85,B 0,C 180,E1 -18978.587,E2 -18978.587} C_VEL
LIN {X 0,Y 249.21,Z 257.443,A -85,B 0,C 180,E1 -18981.895,E2 -18981.895} C_VEL
LIN {X 0,Y 249.361,Z 257.426,A -85,B 0,C 180,E1 -18983.528,E2 -18983.528} C_VEL
LIN {X 0,Y 249.665,Z 257.386,A -85,B 0,C 180,E1 -18988.388,E2 -18988.388} C_VEL
LIN {X 0,Y 249.663,Z 257.386,A -85,B 0,C 180,E1 -18991.614,E2 -18991.614} C_VEL
LIN {X 0,Y 249.448,Z 257.41,A -85,B 0,C 180,E1 -18996.472,E2 -18996.472} C_VEL
LIN {X 0,Y 249.375,Z 257.421,A -85,B 0,C 180,E1 -18999.736,E2 -18999.736} C_VEL
LIN {X 0,Y 249.193,Z 257.446,A -85,B 0,C 180,E1 -19004.705,E2 -19004.705} C_VEL
LIN {X 0,Y 249.138,Z 257.449,A -85,B 0,C 180,E1 -19008.078,E2 -19008.078} C_VEL
LIN {X 0,Y 249.13,Z 257.453,A -85,B 0,C 180,E1 -19011.515,E2 -19011.515} C_VEL
LIN {X 0,Y 249.127,Z 257.45,A -85,B 0,C 180,E1 -19015.488,E2 -19015.488} C_VEL
LIN {X 0,Y 249.073,Z 257.461,A -85,B 0,C 180,E1 -19018.996,E2 -19018.996} C_VEL
LIN {X 0,Y 249.026,Z 257.467,A -85,B 0,C 180,E1 -19022.427,E2 -19022.427} C_VEL
LIN {X 0,Y 249.065,Z 257.456,A -85,B 0,C 180,E1 -19026.34,E2 -19026.34} C_VEL
LIN {X 0,Y 249.075,Z 257.46,A -85,B 0,C 180,E1 -19030.465,E2 -19030.465} C_VEL
LIN {X 0,Y 249.087,Z 257.457,A -85,B 0,C 180,E1 -19032.817,E2 -19032.817} C_VEL
LIN {X 0,Y 249.091,Z 257.446,A -85,B 0,C 180,E1 -19037.383,E2 -19037.383} C_VEL
LIN {X 0,Y 249.048,Z 257.46,A -85,B 0,C 180,E1 -19041.627,E2 -19041.627} C_VEL
LIN {X 0,Y 249.057,Z 257.459,A -85,B 0,C 180,E1 -19045.645,E2 -19045.645} C_VEL
LIN {X 0,Y 249.047,Z 257.453,A -85,B 0,C 180,E1 -19049.476,E2 -19049.476} C_VEL
LIN {X 0,Y 249.07,Z 257.455,A -85,B 0,C 180,E1 -19053.165,E2 -19053.165} C_VEL
LIN {X 0,Y 249.078,Z 257.457,A -85,B 0,C 180,E1 -19056.736,E2 -19056.736} C_VEL
LIN {X 0,Y 249.11,Z 257.451,A -85,B 0,C 180,E1 -19060.215,E2 -19060.215} C_VEL
LIN {X 0,Y 249.242,Z 257.429,A -85,B 0,C 180,E1 -19063.625,E2 -19063.625} C_VEL
LIN {X 0,Y 249.245,Z 257.436,A -85,B 0,C 180,E1 -19068.619,E2 -19068.619} C_VEL
LIN {X 0,Y 249.448,Z 257.412,A -85,B 0,C 180,E1 -19071.905,E2 -19071.905} C_VEL
LIN {X 0,Y 249.295,Z 257.422,A -85,B 0,C 180,E1 -19075.151,E2 -19075.151} C_VEL
LIN {X 0,Y 249.679,Z 257.381,A -85,B 0,C 180,E1 -19078.39,E2 -19078.39} C_VEL
LIN {X 0,Y 249.678,Z 257.385,A -85,B 0,C 180,E1 -19081.616,E2 -19081.616} C_VEL
LIN {X 0,Y 249.44,Z 257.404,A -85,B 0,C 180,E1 -19086.474,E2 -19086.474} C_VEL
LIN {X 0,Y 249.348,Z 257.426,A -85,B 0,C 180,E1 -19089.739,E2 -19089.739} C_VEL
LIN {X 0,Y 249.211,Z 257.438,A -85,B 0,C 180,E1 -19094.706,E2 -19094.706} C_VEL
LIN {X 0,Y 249.146,Z 257.448,A -85,B 0,C 180,E1 -19098.079,E2 -19098.079} C_VEL
LIN {X 0,Y 249.094,Z 257.458,A -85,B 0,C 180,E1 -19101.52,E2 -19101.52} C_VEL
LIN {X 0,Y 249.138,Z 257.453,A -85,B 0,C 180,E1 -19105.484,E2 -19105.484} C_VEL
LIN {X 0,Y 249.081,Z 257.459,A -85,B 0,C 180,E1 -19108.991,E2 -19108.991} C_VEL
LIN {X 0,Y 249.016,Z 257.463,A -85,B 0,C 180,E1 -19112.869,E2 -19112.869} C_VEL
LIN {X 0,Y 249.122,Z 257.638,A -85,B 0,C 180,E1 -19117.294,E2 -19117.294} C_VEL
LIN {X 0,Y 249.161,Z 257.785,A -85,B 0,C 180,E1 -19117.445,E2 -19117.445} C_VEL
LIN {X 0,Y 249.066,Z 258.71,A -85,B 0,C 180,E1 -19118.323,E2 -19118.323} C_VEL
LIN {X 0,Y 247.999,Z 260.265,A -85,B 0,C 180,E1 -19119.618,E2 -19119.618} C_VEL
LIN {X 0,Y 244.208,Z 264.146,A -85,B 0,C 180,E1 -19122.623,E2 -19122.623} C_VEL
LIN {X 0,Y 243.396,Z 265.738,A -85,B 0,C 180,E1 -19123.966,E2 -19123.966} C_VEL
LIN {X 0,Y 243.397,Z 266.235,A -85,B 0,C 180,E1 -19124.421,E2 -19124.421} C_VEL
LIN {X 0,Y 244.298,Z 270.808,A -85,B 0,C 180,E1 -19128.572,E2 -19128.572} C_VEL
LIN {X 0,Y 244.836,Z 274.695,A -85,B 0,C 180,E1 -19131.901,E2 -19131.901} C_VEL
LIN {X 0,Y 244.721,Z 276.689,A -85,B 0,C 180,E1 -19133.528,E2 -19133.528} C_VEL
LIN {X 0,Y 243.82,Z 280.893,A -85,B 0,C 180,E1 -19136.792,E2 -19136.792} C_VEL
LIN {X 0,Y 242.616,Z 286.979,A -85,B 0,C 180,E1 -19141.448,E2 -19141.448} C_VEL
LIN {X 0,Y 242.586,Z 287.093,A -85,B 0,C 180,E1 -19141.534,E2 -19141.534} C_VEL
LIN {X 0,Y 244.965,Z 300.809,A -85,B 0,C 180,E1 -19142.559,E2 -19142.559} C_VEL
LIN {X 0,Y 246.641,Z 312.865,A -85,B 0,C 180,E1 -19143.728,E2 -19143.728} C_VEL
LIN {X 0,Y 247.79,Z 325.049,A -85,B 0,C 180,E1 -19145.181,E2 -19145.181} C_VEL
LIN {X 0,Y 248.439,Z 336.785,A -85,B 0,C 180,E1 -19146.889,E2 -19146.889} C_VEL
LIN {X 0,Y 248.413,Z 342.051,A -85,B 0,C 180,E1 -19147.765,E2 -19147.765} C_VEL
LIN {X 0,Y 246.526,Z 351.847,A -85,B 0,C 180,E1 -19149.559,E2 -19149.559} C_VEL
LIN {X 0,Y 244.797,Z 360.807,A -85,B 0,C 180,E1 -19151.59,E2 -19151.59} C_VEL
LIN {X 0,Y 243.349,Z 368.222,A -85,B 0,C 180,E1 -19153.644,E2 -19153.644} C_VEL
LIN {X 0,Y 241.948,Z 375.514,A -85,B 0,C 180,E1 -19156.134,E2 -19156.134} C_VEL
LIN {X 0,Y 241.125,Z 380.448,A -85,B 0,C 180,E1 -19158.227,E2 -19158.227} C_VEL
LIN {X 0,Y 240.489,Z 385.229,A -85,B 0,C 180,E1 -19160.75,E2 -19160.75} C_VEL
LIN {X 0,Y 240.136,Z 388.865,A -85,B 0,C 180,E1 -19163.276,E2 -19163.276} C_VEL
LIN {X 0,Y 240.065,Z 390.73,A -85,B 0,C 180,E1 -19164.961,E2 -19164.961} C_VEL
LIN {X 0,Y 240.061,Z 392.115,A -85,B 0,C 180,E1 -19166.642,E2 -19166.642} C_VEL
LIN {X 0,Y 240.04,Z 393.073,A -85,B 0,C 180,E1 -19168.321,E2 -19168.321} C_VEL
LIN {X 0,Y 240.101,Z 393.633,A -85,B 0,C 180,E1 -19169.999,E2 -19169.999} C_VEL
LIN {X 0,Y 240.031,Z 393.782,A -85,B 0,C 180,E1 -19171.677,E2 -19171.677} C_VEL
LIN {X 0,Y 239.998,Z 393.49,A -85,B 0,C 180,E1 -19173.357,E2 -19173.357} C_VEL
LIN {X 0,Y 239.994,Z 392.648,A -85,B 0,C 180,E1 -19175.32,E2 -19175.32} C_VEL
LIN {X 0,Y 240.269,Z 390.247,A -85,B 0,C 180,E1 -19178.409,E2 -19178.409} C_VEL
LIN {X 0,Y 240.853,Z 387.211,A -85,B 0,C 180,E1 -19180.932,E2 -19180.932} C_VEL
LIN {X 0,Y 241.795,Z 383.172,A -85,B 0,C 180,E1 -19183.445,E2 -19183.445} C_VEL
LIN {X 0,Y 243.36,Z 378.043,A -85,B 0,C 180,E1 -19185.922,E2 -19185.922} C_VEL
LIN {X 0,Y 245.245,Z 371.673,A -85,B 0,C 180,E1 -19188.374,E2 -19188.374} C_VEL
LIN {X 0,Y 247.448,Z 363.834,A -85,B 0,C 180,E1 -19190.794,E2 -19190.794} C_VEL
LIN {X 0,Y 250.265,Z 354.178,A -85,B 0,C 180,E1 -19193.15,E2 -19193.15} C_VEL
LIN {X 0,Y 252.368,Z 346.426,A -85,B 0,C 180,E1 -19194.69,E2 -19194.69} C_VEL
LIN {X 0,Y 253.298,Z 335.871,A -85,B 0,C 180,E1 -19196.637,E2 -19196.637} C_VEL
LIN {X 0,Y 253.389,Z 326.71,A -85,B 0,C 180,E1 -19198.131,E2 -19198.131} C_VEL
LIN {X 0,Y 252.465,Z 315.4,A -85,B 0,C 180,E1 -19199.859,E2 -19199.859} C_VEL
LIN {X 0,Y 250.577,Z 304.395,A -85,B 0,C 180,E1 -19201.431,E2 -19201.431} C_VEL
LIN {X 0,Y 247.227,Z 291.935,A -85,B 0,C 180,E1 -19203.178,E2 -19203.178} C_VEL
LIN {X 0,Y 245.396,Z 286.842,A -85,B 0,C 180,E1 -19203.914,E2 -19203.914} C_VEL
LIN {X 0,Y 244.589,Z 283.621,A -85,B 0,C 180,E1 -19204.312,E2 -19204.312} C_VEL
LIN {X 0,Y 245.284,Z 280.501,A -85,B 0,C 180,E1 -19206.991,E2 -19206.991} C_VEL
LIN {X 0,Y 245.405,Z 278.003,A -85,B 0,C 180,E1 -19209.351,E2 -19209.351} C_VEL
LIN {X 0,Y 245.124,Z 275.61,A -85,B 0,C 180,E1 -19211.799,E2 -19211.799} C_VEL
LIN {X 0,Y 244.34,Z 271.633,A -85,B 0,C 180,E1 -19216.342,E2 -19216.342} C_VEL
LIN {X 0,Y 243.818,Z 268.345,A -85,B 0,C 180,E1 -19220.641,E2 -19220.641} C_VEL
LIN {X 0,Y 243.34,Z 265.697,A -85,B 0,C 180,E1 -19224.713,E2 -19224.713} C_VEL
LIN {X 0,Y 242.942,Z 263.588,A -85,B 0,C 180,E1 -19228.617,E2 -19228.617} C_VEL
LIN {X 0,Y 242.674,Z 261.934,A -85,B 0,C 180,E1 -19232.393,E2 -19232.393} C_VEL
LIN {X 0,Y 242.476,Z 260.702,A -85,B 0,C 180,E1 -19236.057,E2 -19236.057} C_VEL
LIN {X 0,Y 242.339,Z 259.84,A -85,B 0,C 180,E1 -19239.632,E2 -19239.632} C_VEL
LIN {X 0,Y 242.337,Z 259.295,A -85,B 0,C 180,E1 -19243.139,E2 -19243.139} C_VEL
LIN {X 0,Y 242.326,Z 259.054,A -85,B 0,C 180,E1 -19248.284,E2 -19248.284} C_VEL
LIN {X 0,Y 242.583,Z 259.187,A -85,B 0,C 180,E1 -19251.668,E2 -19251.668} C_VEL
LIN {X 0,Y 242.69,Z 259.916,A -85,B 0,C 180,E1 -19256.677,E2 -19256.677} C_VEL
LIN {X 0,Y 243.117,Z 260.604,A -85,B 0,C 180,E1 -19259.997,E2 -19259.997} C_VEL
LIN {X 0,Y 242.967,Z 261.616,A -85,B 0,C 180,E1 -19263.314,E2 -19263.314} C_VEL
LIN {X 0,Y 243.086,Z 262.87,A -85,B 0,C 180,E1 -19266.89,E2 -19266.89} C_VEL
LIN {X 0,Y 243.044,Z 264.365,A -85,B 0,C 180,E1 -19270.535,E2 -19270.535} C_VEL
LIN {X 0,Y 242.904,Z 265.458,A -85,B 0,C 180,E1 -19272.53,E2 -19272.53} C_VEL
LIN {X 0,Y 244.046,Z 268.381,A -85,B 0,C 180,E1 -19272.999,E2 -19272.999} C_VEL
LIN {X 0,Y 245.432,Z 270.548,A -85,B 0,C 180,E1 -19273.468,E2 -19273.468} C_VEL
LIN {X 0,Y 250.368,Z 281.191,A -85,B 0,C 180,E1 -19275.463,E2 -19275.463} C_VEL
LIN {X 0,Y 254.062,Z 291.657,A -85,B 0,C 180,E1 -19277.379,E2 -19277.379} C_VEL
LIN {X 0,Y 256.445,Z 301.6,A -85,B 0,C 180,E1 -19279.197,E2 -19279.197} C_VEL
LIN {X 0,Y 257.612,Z 309.87,A -85,B 0,C 180,E1 -19280.769,E2 -19280.769} C_VEL
LIN {X 0,Y 255.145,Z 320.467,A -85,B 0,C 180,E1 -19282.516,E2 -19282.516} C_VEL
LIN {X 0,Y 252.557,Z 329.841,A -85,B 0,C 180,E1 -19284.425,E2 -19284.425} C_VEL
LIN {X 0,Y 249.878,Z 338.894,A -85,B 0,C 180,E1 -19286.741,E2 -19286.741} C_VEL
LIN {X 0,Y 247.256,Z 346.842,A -85,B 0,C 180,E1 -19289.358,E2 -19289.358} C_VEL
LIN {X 0,Y 245.113,Z 353.12,A -85,B 0,C 180,E1 -19292.03,E2 -19292.03} C_VEL
LIN {X 0,Y 243.642,Z 357.216,A -85,B 0,C 180,E1 -19294.289,E2 -19294.289} C_VEL
LIN {X 0,Y 242.371,Z 360.516,A -85,B 0,C 180,E1 -19296.645,E2 -19296.645} C_VEL
LIN {X 0,Y 241.698,Z 362.267,A -85,B 0,C 180,E1 -19298.272,E2 -19298.272} C_VEL
LIN {X 0,Y 240.884,Z 364.074,A -85,B 0,C 180,E1 -19300.663,E2 -19300.663} C_VEL
LIN {X 0,Y 240.323,Z 365.046,A -85,B 0,C 180,E1 -19303.023,E2 -19303.023} C_VEL
LIN {X 0,Y 240.019,Z 365.242,A -85,B 0,C 180,E1 -19305.354,E2 -19305.354} C_VEL
LIN {X 0,Y 239.909,Z 364.671,A -85,B 0,C 180,E1 -19307.643,E2 -19307.643} C_VEL
LIN {X 0,Y 240.038,Z 363.357,A -85,B 0,C 180,E1 -19309.901,E2 -19309.901} C_VEL
LIN {X 0,Y 240.595,Z 360.101,A -85,B 0,C 180,E1 -19313.216,E2 -19313.216} C_VEL
LIN {X 0,Y 241.171,Z 356.683,A -85,B 0,C 180,E1 -19315.588,E2 -19315.588} C_VEL
LIN {X 0,Y 242.191,Z 351.035,A -85,B 0,C 180,E1 -19318.512,E2 -19318.512} C_VEL
LIN {X 0,Y 243.432,Z 344.612,A -85,B 0,C 180,E1 -19321.082,E2 -19321.082} C_VEL
LIN {X 0,Y 244.984,Z 336.695,A -85,B 0,C 180,E1 -19323.6,E2 -19323.6} C_VEL
LIN {X 0,Y 246.629,Z 328.187,A -85,B 0,C 180,E1 -19325.758,E2 -19325.758} C_VEL
LIN {X 0,Y 248.374,Z 318.447,A -85,B 0,C 180,E1 -19327.763,E2 -19327.763} C_VEL
LIN {X 0,Y 250.313,Z 306.815,A -85,B 0,C 180,E1 -19329.67,E2 -19329.67} C_VEL
LIN {X 0,Y 251.036,Z 300.166,A -85,B 0,C 180,E1 -19330.583,E2 -19330.583} C_VEL
LIN {X 0,Y 248.939,Z 289.041,A -85,B 0,C 180,E1 -19332.145,E2 -19332.145} C_VEL
LIN {X 0,Y 246.421,Z 278.289,A -85,B 0,C 180,E1 -19333.43,E2 -19333.43} C_VEL
LIN {X 0,Y 242.79,Z 265.782,A -85,B 0,C 180,E1 -19334.688,E2 -19334.688} C_VEL
LIN {X 0,Y 241.271,Z 260.748,A -85,B 0,C 180,E1 -19335.127,E2 -19335.127} C_VEL
LIN {X 0,Y 241.496,Z 258.482,A -85,B 0,C 180,E1 -19338.247,E2 -19338.247} C_VEL
LIN {X 0,Y 242.118,Z 258.328,A -85,B 0,C 180,E1 -19341.656,E2 -19341.656} C_VEL
LIN {X 0,Y 242.296,Z 258.306,A -85,B 0,C 180,E1 -19343.338,E2 -19343.338} C_VEL
LIN {X 0,Y 242.625,Z 258.263,A -85,B 0,C 180,E1 -19348.341,E2 -19348.341} C_VEL
LIN {X 0,Y 242.623,Z 258.262,A -85,B 0,C 180,E1 -19351.661,E2 -19351.661} C_VEL
LIN {X 0,Y 242.42,Z 258.286,A -85,B 0,C 180,E1 -19356.66,E2 -19356.66} C_VEL
LIN {X 0,Y 242.301,Z 258.302,A -85,B 0,C 180,E1 -19360.023,E2 -19360.023} C_VEL
LIN {X 0,Y 242.154,Z 258.325,A -85,B 0,C 180,E1 -19365.142,E2 -19365.142} C_VEL
LIN {X 0,Y 242.08,Z 258.33,A -85,B 0,C 180,E1 -19368.624,E2 -19368.624} C_VEL
LIN {X 0,Y 242.062,Z 258.334,A -85,B 0,C 180,E1 -19372.176,E2 -19372.176} C_VEL
LIN {X 0,Y 242.055,Z 258.33,A -85,B 0,C 180,E1 -19375.84,E2 -19375.84} C_VEL
LIN {X 0,Y 242.02,Z 258.337,A -85,B 0,C 180,E1 -19379.582,E2 -19379.582} C_VEL
LIN {X 0,Y 241.981,Z 258.34,A -85,B 0,C 180,E1 -19383.493,E2 -19383.493} C_VEL
LIN {X 0,Y 242.003,Z 258.334,A -85,B 0,C 180,E1 -19387.58,E2 -19387.58} C_VEL
LIN {X 0,Y 242.03,Z 258.335,A -85,B 0,C 180,E1 -19391.904,E2 -19391.904} C_VEL
LIN {X 0,Y 242.017,Z 258.331,A -85,B 0,C 180,E1 -19396.552,E2 -19396.552} C_VEL
LIN {X 0,Y 242.005,Z 258.337,A -85,B 0,C 180,E1 -19400.295,E2 -19400.295} C_VEL
LIN {X 0,Y 242.032,Z 258.337,A -85,B 0,C 180,E1 -19404.501,E2 -19404.501} C_VEL
LIN {X 0,Y 241.972,Z 258.336,A -85,B 0,C 180,E1 -19408.483,E2 -19408.483} C_VEL
LIN {X 0,Y 242.004,Z 258.336,A -85,B 0,C 180,E1 -19412.316,E2 -19412.316} C_VEL
LIN {X 0,Y 242.055,Z 258.334,A -85,B 0,C 180,E1 -19416.019,E2 -19416.019} C_VEL
LIN {X 0,Y 242.036,Z 258.333,A -85,B 0,C 180,E1 -19419.611,E2 -19419.611} C_VEL
LIN {X 0,Y 242.163,Z 258.308,A -85,B 0,C 180,E1 -19423.281,E2 -19423.281} C_VEL
LIN {X 0,Y 242.182,Z 258.318,A -85,B 0,C 180,E1 -19428.283,E2 -19428.283} C_VEL
LIN {X 0,Y 242.395,Z 258.291,A -85,B 0,C 180,E1 -19431.667,E2 -19431.667} C_VEL
LIN {X 0,Y 242.255,Z 258.298,A -85,B 0,C 180,E1 -19435.01,E2 -19435.01} C_VEL
LIN {X 0,Y 242.639,Z 258.258,A -85,B 0,C 180,E1 -19438.343,E2 -19438.343} C_VEL
LIN {X 0,Y 242.638,Z 258.263,A -85,B 0,C 180,E1 -19441.663,E2 -19441.663} C_VEL
LIN {X 0,Y 242.411,Z 258.279,A -85,B 0,C 180,E1 -19446.662,E2 -19446.662} C_VEL
LIN {X 0,Y 242.272,Z 258.306,A -85,B 0,C 180,E1 -19450.026,E2 -19450.026} C_VEL
LIN {X 0,Y 242.173,Z 258.316,A -85,B 0,C 180,E1 -19455.143,E2 -19455.143} C_VEL
LIN {X 0,Y 242.08,Z 258.327,A -85,B 0,C 180,E1 -19458.626,E2 -19458.626} C_VEL
LIN {X 0,Y 242.02,Z 258.336,A -85,B 0,C 180,E1 -19462.182,E2 -19462.182} C_VEL
LIN {X 0,Y 242.074,Z 258.331,A -85,B 0,C 180,E1 -19465.84,E2 -19465.84} C_VEL
LIN {X 0,Y 242.015,Z 258.34,A -85,B 0,C 180,E1 -19469.585,E2 -19469.585} C_VEL
LIN {X 0,Y 241.989,Z 258.343,A -85,B 0,C 180,E1 -19473.494,E2 -19473.494} C_VEL
LIN {X 0,Y 242.069,Z 258.478,A -85,B 0,C 180,E1 -19476.786,E2 -19476.786} C_VEL
LIN {X 0,Y 242.813,Z 262.837,A -85,B 0,C 180,E1 -19481.187,E2 -19481.187} C_VEL
LIN {X 0,Y 243.397,Z 266.235,A -85,B 0,C 180,E1 -19484.421,E2 -19484.421} C_VEL
LIN {X 0,Y 242.996,Z 267.781,A -85,B 0,C 180,E1 -19485.759,E2 -19485.759} C_VEL
LIN {X 0,Y 240.592,Z 270.613,A -85,B 0,C 180,E1 -19487.939,E2 -19487.939} C_VEL
LIN {X 0,Y 238.531,Z 272.944,A -85,B 0,C 180,E1 -19489.708,E2 -19489.708} C_VEL
LIN {X 0,Y 237.764,Z 274.638,A -85,B 0,C 180,E1 -19491.075,E2 -19491.075} C_VEL
LIN {X 0,Y 237.77,Z 275.178,A -85,B 0,C 180,E1 -19491.538,E2 -19491.538} C_VEL
LIN {X 0,Y 237.59,Z 277.787,A -85,B 0,C 180,E1 -19493.728,E2 -19493.728} C_VEL
LIN {X 0,Y 236.498,Z 282.679,A -85,B 0,C 180,E1 -19497.662,E2 -19497.662} C_VEL
LIN {X 0,Y 235.667,Z 286.713,A -85,B 0,C 180,E1 -19500.836,E2 -19500.836} C_VEL
LIN {X 0,Y 238.079,Z 300.79,A -85,B 0,C 180,E1 -19501.935,E2 -19501.935} C_VEL
LIN {X 0,Y 239.858,Z 313.544,A -85,B 0,C 180,E1 -19503.241,E2 -19503.241} C_VEL
LIN {X 0,Y 240.915,Z 325.554,A -85,B 0,C 180,E1 -19504.738,E2 -19504.738} C_VEL
LIN {X 0,Y 241.515,Z 336.635,A -85,B 0,C 180,E1 -19506.413,E2 -19506.413} C_VEL
LIN {X 0,Y 241.401,Z 343.079,A -85,B 0,C 180,E1 -19507.534,E2 -19507.534} C_VEL
LIN {X 0,Y 239.43,Z 352.622,A -85,B 0,C 180,E1 -19509.375,E2 -19509.375} C_VEL
LIN {X 0,Y 237.702,Z 361.39,A -85,B 0,C 180,E1 -19511.467,E2 -19511.467} C_VEL
LIN {X 0,Y 236.221,Z 368.635,A -85,B 0,C 180,E1 -19513.581,E2 -19513.581} C_VEL
LIN {X 0,Y 234.796,Z 375.76,A -85,B 0,C 180,E1 -19516.145,E2 -19516.145} C_VEL
LIN {X 0,Y 233.868,Z 381.44,A -85,B 0,C 180,E1 -19518.735,E2 -19518.735} C_VEL
LIN {X 0,Y 233.272,Z 385.893,A -85,B 0,C 180,E1 -19521.335,E2 -19521.335} C_VEL
LIN {X 0,Y 233.037,Z 389.736,A -85,B 0,C 180,E1 -19524.418,E2 -19524.418} C_VEL
LIN {X 0,Y 232.977,Z 391.576,A -85,B 0,C 180,E1 -19526.54,E2 -19526.54} C_VEL
LIN {X 0,Y 232.971,Z 392.565,A -85,B 0,C 180,E1 -19528.27,E2 -19528.27} C_VEL
LIN {X 0,Y 233.026,Z 393.155,A -85,B 0,C 180,E1 -19529.999,E2 -19529.999} C_VEL
LIN {X 0,Y 232.96,Z 393.336,A -85,B 0,C 180,E1 -19531.728,E2 -19531.728} C_VEL
LIN {X 0,Y 232.915,Z 393.105,A -85,B 0,C 180,E1 -19533.459,E2 -19533.459} C_VEL
LIN {X 0,Y 232.921,Z 392.399,A -85,B 0,C 180,E1 -19535.28,E2 -19535.28} C_VEL
LIN {X 0,Y 233.225,Z 389.955,A -85,B 0,C 180,E1 -19538.665,E2 -19538.665} C_VEL
LIN {X 0,Y 233.868,Z 386.984,A -85,B 0,C 180,E1 -19541.263,E2 -19541.263} C_VEL
LIN {X 0,Y 234.862,Z 383.02,A -85,B 0,C 180,E1 -19543.85,E2 -19543.85} C_VEL
LIN {X 0,Y 236.521,Z 377.99,A -85,B 0,C 180,E1 -19546.395,E2 -19546.395} C_VEL
LIN {X 0,Y 238.517,Z 371.74,A -85,B 0,C 180,E1 -19548.911,E2 -19548.911} C_VEL
LIN {X 0,Y 240.807,Z 364.063,A -85,B 0,C 180,E1 -19551.395,E2 -19551.395} C_VEL
LIN {X 0,Y 243.777,Z 354.54,A -85,B 0,C 180,E1 -19553.803,E2 -19553.803} C_VEL
LIN {X 0,Y 245.907,Z 346.95,A -85,B 0,C 180,E1 -19555.384,E2 -19555.384} C_VEL
LIN {X 0,Y 247.058,Z 335.115,A -85,B 0,C 180,E1 -19557.657,E2 -19557.657} C_VEL
LIN {X 0,Y 247.079,Z 324.695,A -85,B 0,C 180,E1 -19559.435,E2 -19559.435} C_VEL
LIN {X 0,Y 245.778,Z 312.377,A -85,B 0,C 180,E1 -19561.383,E2 -19561.383} C_VEL
LIN {X 0,Y 243.46,Z 300.713,A -85,B 0,C 180,E1 -19563.156,E2 -19563.156} C_VEL
LIN {X 0,Y 240.439,Z 290.682,A -85,B 0,C 180,E1 -19564.701,E2 -19564.701} C_VEL
LIN {X 0,Y 239.245,Z 287.126,A -85,B 0,C 180,E1 -19565.231,E2 -19565.231} C_VEL
LIN {X 0,Y 238.055,Z 283.645,A -85,B 0,C 180,E1 -19565.753,E2 -19565.753} C_VEL
LIN {X 0,Y 238,Z 282.931,A -85,B 0,C 180,E1 -19565.904,E2 -19565.904} C_VEL
LIN {X 0,Y 238.456,Z 280.425,A -85,B 0,C 180,E1 -19568.237,E2 -19568.237} C_VEL
LIN {X 0,Y 238.265,Z 278.24,A -85,B 0,C 180,E1 -19570.459,E2 -19570.459} C_VEL
LIN {X 0,Y 237.964,Z 276.115,A -85,B 0,C 180,E1 -19572.786,E2 -19572.786} C_VEL
LIN {X 0,Y 237.302,Z 272.564,A -85,B 0,C 180,E1 -19577.062,E2 -19577.062} C_VEL
LIN {X 0,Y 236.804,Z 269.388,A -85,B 0,C 180,E1 -19581.443,E2 -19581.443} C_VEL
LIN {X 0,Y 236.314,Z 266.866,A -85,B 0,C 180,E1 -19585.591,E2 -19585.591} C_VEL
LIN {X 0,Y 235.954,Z 264.772,A -85,B 0,C 180,E1 -19589.741,E2 -19589.741} C_VEL
LIN {X 0,Y 235.762,Z 263.277,A -85,B 0,C 180,E1 -19593.437,E2 -19593.437} C_VEL
LIN {X 0,Y 235.509,Z 262.024,A -85,B 0,C 180,E1 -19597.679,E2 -19597.679} C_VEL
LIN {X 0,Y 235.45,Z 261.095,A -85,B 0,C 180,E1 -19602.776,E2 -19602.776} C_VEL
LIN {X 0,Y 235.412,Z 260.803,A -85,B 0,C 180,E1 -19606.18,E2 -19606.18} C_VEL
LIN {X 0,Y 235.597,Z 260.769,A -85,B 0,C 180,E1 -19609.862,E2 -19609.862} C_VEL
LIN {X 0,Y 235.689,Z 261.021,A -85,B 0,C 180,E1 -19613.147,E2 -19613.147} C_VEL
LIN {X 0,Y 236.021,Z 261.809,A -85,B 0,C 180,E1 -19618.291,E2 -19618.291} C_VEL
LIN {X 0,Y 236.2,Z 262.168,A -85,B 0,C 180,E1 -19619.997,E2 -19619.997} C_VEL
LIN {X 0,Y 236.04,Z 263.176,A -85,B 0,C 180,E1 -19623.411,E2 -19623.411} C_VEL
LIN {X 0,Y 236.152,Z 264.327,A -85,B 0,C 180,E1 -19626.868,E2 -19626.868} C_VEL
LIN {X 0,Y 236.066,Z 266.01,A -85,B 0,C 180,E1 -19630.906,E2 -19630.906} C_VEL
LIN {X 0,Y 237.061,Z 268.764,A -85,B 0,C 180,E1 -19631.373,E2 -19631.373} C_VEL
LIN {X 0,Y 238.608,Z 271.118,A -85,B 0,C 180,E1 -19631.949,E2 -19631.949} C_VEL
LIN {X 0,Y 242.621,Z 279.2,A -85,B 0,C 180,E1 -19633.637,E2 -19633.637} C_VEL
LIN {X 0,Y 246.694,Z 289.503,A -85,B 0,C 180,E1 -19635.699,E2 -19635.699} C_VEL
LIN {X 0,Y 249.437,Z 299.205,A -85,B 0,C 180,E1 -19637.597,E2 -19637.597} C_VEL
LIN {X 0,Y 251.274,Z 310.362,A -85,B 0,C 180,E1 -19639.821,E2 -19639.821} C_VEL
LIN {X 0,Y 251.19,Z 312.667,A -85,B 0,C 180,E1 -19640.254,E2 -19640.254} C_VEL
LIN {X 0,Y 248.587,Z 322.693,A -85,B 0,C 180,E1 -19641.995,E2 -19641.995} C_VEL
LIN {X 0,Y 245.98,Z 331.537,A -85,B 0,C 180,E1 -19643.899,E2 -19643.899} C_VEL
LIN {X 0,Y 243.12,Z 340.513,A -85,B 0,C 180,E1 -19646.348,E2 -19646.348} C_VEL
LIN {X 0,Y 240.601,Z 347.644,A -85,B 0,C 180,E1 -19648.803,E2 -19648.803} C_VEL
LIN {X 0,Y 238.532,Z 353.358,A -85,B 0,C 180,E1 -19651.304,E2 -19651.304} C_VEL
LIN {X 0,Y 236.821,Z 357.803,A -85,B 0,C 180,E1 -19653.807,E2 -19653.807} C_VEL
LIN {X 0,Y 235.281,Z 361.586,A -85,B 0,C 180,E1 -19656.681,E2 -19656.681} C_VEL
LIN {X 0,Y 234.335,Z 363.701,A -85,B 0,C 180,E1 -19659.032,E2 -19659.032} C_VEL
LIN {X 0,Y 233.582,Z 365.077,A -85,B 0,C 180,E1 -19661.443,E2 -19661.443} C_VEL
LIN {X 0,Y 233.115,Z 365.683,A -85,B 0,C 180,E1 -19663.896,E2 -19663.896} C_VEL
LIN {X 0,Y 232.853,Z 365.478,A -85,B 0,C 180,E1 -19666.411,E2 -19666.411} C_VEL
LIN {X 0,Y 232.859,Z 364.375,A -85,B 0,C 180,E1 -19668.979,E2 -19668.979} C_VEL
LIN {X 0,Y 233.172,Z 362.319,A -85,B 0,C 180,E1 -19671.591,E2 -19671.591} C_VEL
LIN {X 0,Y 233.73,Z 359.192,A -85,B 0,C 180,E1 -19674.272,E2 -19674.272} C_VEL
LIN {X 0,Y 234.643,Z 354.124,A -85,B 0,C 180,E1 -19677.377,E2 -19677.377} C_VEL
LIN {X 0,Y 235.859,Z 347.756,A -85,B 0,C 180,E1 -19680.298,E2 -19680.298} C_VEL
LIN {X 0,Y 237.254,Z 341.108,A -85,B 0,C 180,E1 -19682.699,E2 -19682.699} C_VEL
LIN {X 0,Y 238.955,Z 332.443,A -85,B 0,C 180,E1 -19685.206,E2 -19685.206} C_VEL
LIN {X 0,Y 240.907,Z 322.525,A -85,B 0,C 180,E1 -19687.488,E2 -19687.488} C_VEL
LIN {X 0,Y 242.812,Z 311.665,A -85,B 0,C 180,E1 -19689.48,E2 -19689.48} C_VEL
LIN {X 0,Y 244.285,Z 302.071,A -85,B 0,C 180,E1 -19690.899,E2 -19690.899} C_VEL
LIN {X 0,Y 242.358,Z 291.235,A -85,B 0,C 180,E1 -19692.492,E2 -19692.492} C_VEL
LIN {X 0,Y 239.664,Z 279.485,A -85,B 0,C 180,E1 -19693.969,E2 -19693.969} C_VEL
LIN {X 0,Y 235.954,Z 266.619,A -85,B 0,C 180,E1 -19695.335,E2 -19695.335} C_VEL
LIN {X 0,Y 234.277,Z 261.114,A -85,B 0,C 180,E1 -19695.894,E2 -19695.894} C_VEL
LIN {X 0,Y 234.419,Z 259.704,A -85,B 0,C 180,E1 -19697.887,E2 -19697.887} C_VEL
LIN {X 0,Y 234.92,Z 259.222,A -85,B 0,C 180,E1 -19700.816,E2 -19700.816} C_VEL
LIN {X 0,Y 235.213,Z 259.188,A -85,B 0,C 180,E1 -19703.137,E2 -19703.137} C_VEL
LIN {X 0,Y 235.584,Z 259.14,A -85,B 0,C 180,E1 -19708.291,E2 -19708.291} C_VEL
LIN {X 0,Y 235.583,Z 259.139,A -85,B 0,C 180,E1 -19711.71,E2 -19711.71} C_VEL
LIN {X 0,Y 235.391,Z 259.162,A -85,B 0,C 180,E1 -19716.86,E2 -19716.86} C_VEL
LIN {X 0,Y 235.225,Z 259.183,A -85,B 0,C 180,E1 -19720.328,E2 -19720.328} C_VEL
LIN {X 0,Y 235.101,Z 259.201,A -85,B 0,C 180,E1 -19725.608,E2 -19725.608} C_VEL
LIN {X 0,Y 235.023,Z 259.21,A -85,B 0,C 180,E1 -19729.205,E2 -19729.205} C_VEL
LIN {X 0,Y 234.993,Z 259.218,A -85,B 0,C 180,E1 -19732.88,E2 -19732.88} C_VEL
LIN {X 0,Y 234.959,Z 259.215,A -85,B 0,C 180,E1 -19736.659,E2 -19736.659} C_VEL
LIN {X 0,Y 234.922,Z 259.224,A -85,B 0,C 180,E1 -19740.57,E2 -19740.57} C_VEL
LIN {X 0,Y 234.951,Z 259.216,A -85,B 0,C 180,E1 -19744.635,E2 -19744.635} C_VEL
LIN {X 0,Y 234.958,Z 259.216,A -85,B 0,C 180,E1 -19748.955,E2 -19748.955} C_VEL
LIN {X 0,Y 234.989,Z 259.211,A -85,B 0,C 180,E1 -19753.463,E2 -19753.463} C_VEL
LIN {X 0,Y 234.989,Z 259.205,A -85,B 0,C 180,E1 -19756.542,E2 -19756.542} C_VEL
LIN {X 0,Y 234.965,Z 259.214,A -85,B 0,C 180,E1 -19761.092,E2 -19761.092} C_VEL
LIN {X 0,Y 234.956,Z 259.215,A -85,B 0,C 180,E1 -19765.37,E2 -19765.37} C_VEL
LIN {X 0,Y 234.965,Z 259.207,A -85,B 0,C 180,E1 -19770.161,E2 -19770.161} C_VEL
LIN {X 0,Y 234.992,Z 259.21,A -85,B 0,C 180,E1 -19773.797,E2 -19773.797} C_VEL
LIN {X 0,Y 235.01,Z 259.207,A -85,B 0,C 180,E1 -19778.973,E2 -19778.973} C_VEL
LIN {X 0,Y 235.096,Z 259.188,A -85,B 0,C 180,E1 -19783.063,E2 -19783.063} C_VEL
LIN {X 0,Y 235.116,Z 259.199,A -85,B 0,C 180,E1 -19787.925,E2 -19787.925} C_VEL
LIN {X 0,Y 235.327,Z 259.17,A -85,B 0,C 180,E1 -19791.415,E2 -19791.415} C_VEL
LIN {X 0,Y 235.369,Z 259.161,A -85,B 0,C 180,E1 -19793.143,E2 -19793.143} C_VEL
LIN {X 0,Y 235.598,Z 259.135,A -85,B 0,C 180,E1 -19798.293,E2 -19798.293} C_VEL
LIN {X 0,Y 235.598,Z 259.14,A -85,B 0,C 180,E1 -19801.712,E2 -19801.712} C_VEL
LIN {X 0,Y 235.363,Z 259.157,A -85,B 0,C 180,E1 -19806.863,E2 -19806.863} C_VEL
LIN {X 0,Y 235.219,Z 259.183,A -85,B 0,C 180,E1 -19810.33,E2 -19810.33} C_VEL
LIN {X 0,Y 235.12,Z 259.193,A -85,B 0,C 180,E1 -19815.609,E2 -19815.609} C_VEL
LIN {X 0,Y 235.016,Z 259.21,A -85,B 0,C 180,E1 -19819.208,E2 -19819.208} C_VEL
